(* Version history:
Date	|	Version/Author |	Remark
----------------------------------------------------------------------------------------------------
11.09.01	|	2.01 JP		|	new version depending on 0.99D
22.11.01	|	2.02 JP		|	new version depending on 0.99F
18.01.02	|	2.03 JP		|	new version depending on 1.0
		|				|	changed names, interfaces, execute behavior
25.01.02	|	2.04 JP		|	no CAMMING, change behavior of MC_Power
07.02.02	|	2.05 JP		|	SetOverride in unit less than 1%
13.02.02	|	2.06 JP		|	New: MC_NewPos and MC_NewPosAndVelo
		|				|	removed MC_MoveAdditive
14.02.02	|	2.07 JP		|	completed: MC_Home, MC_MoveSuperImposed
14.02.02	|	2.08 JP		|	renamed MC_NewPosAndVelo New: MC_SetOverride edge triggered
15.02.02	|	2.09 JP		|	changed: MC_Gear
15.02.02	|	2.10 JP		|	changed: MC_SetOverride
04.04.02	|	2.11 JP		|	changed: done for MC_Home 
		|				|	new: Check TimeOut for MoveAbsolute, MoveRelative, Home
08.03.02	|	2.12 JP		|	changed: new flag inserted 
12.03.02	|	2.13 JP		|	changed: reset of bNotExecute
18.03.02	|	2.14 JP		|	changed: MC_Reset waits for ready
22.03.02	|	2.15 JP		|	changed: MC_Read and Write FBs
26.03.02	|	2.16 JP		|	revised: Read/Write Parameter FBs
27.03.02	|	2.17 JP		|	revised: Read/Write Parameter FBs and Home (calibration cam)
09.04.02	|	2.18 JP		|	changed parameter type of some parameters
17.04.02	|	2.19 JP		|	changed: Read(Bool)Parameter new Input to select read mode
							Boolean parameters can be read with ReadParameter
							changed MC_Power: new input override !!			
23.04.02	|	2.20 JP		|	fixed: MC_Home changed: Behavior of MC_MoveAbsolute/Relative
25.04.02	|	2.21 JP		|	changed: MC_Reset: now not waiting for 'axis is ready'. Check with MC_Power !
26.04.02	|	2.22 JP		|	MC_Home: If Posistion =  DEFAULT_HOME_POSITION --> no set of position
							MC_MoveXX: more detailed error messages
05.07.02	|	2.23 JP		|	new MC_MoveAbsoluteOrRestart: combines MoveAbsolute and NewPos
19.07.02	|	2.24 JP		|	changed: E_STATES ---> E_TCMC_STATES
12.09.02	|	2.25 KST		|	changed: MC_MoveAbsolute and MC_MoveRelative now based on FB_MoveGeneric
							MC_NewPos and MC_NewPosAndVelo based on new FB_NewPosAndVeloGeneric 
							new internal start types in MC_MoveAbsoluteOrRestart (message suppression)
16.09.02	|	2.26 ChristophC|	changed: MC_SetActualPosition due to changes in TcNC.Lib
16.10.02	|	2.27 KST		|	new: MC_ExtSetPointGenEnable and MC_ExtSetPointGenDisable
29.10.02	|	2.28 ChristophC|	MC_Stop and MC_SetActualPosition: Ads port changed from TcMcGlobal.NCPORT_TCMC => AMSPORT_R0_NCSAF
12.11.02	|	2.29 ChristophC|	MC_OverrideFilter function block added
13.12.02	|	2.30 JP		|	several smaller changes: MC_ReadStatus, MC_Stop
22.01.03	|	2.31 KSt		|	new additional function MC_ExtSetPointGenFeed
24.03.03	|	2.32 JP		|	added: MC_GearFloat, corr. MC_ReadBoolParameter (wrong for AxisEnPostionRangeMonitoring)
26.03.03	|	2.33 KSt		|	added: MC_MoveModulo
04.04.03	|	2.34 KSt		|	changed: MC_MoveAbsoluteOrRestart, Done will be reset at once after Execute=FALSE
12.05.03	|	2.35 JP		|	changed: MC_MoveVelocity, MC_Home (error handling), MC_ReadStatus
14.05.03	|	2.36 KSt		|	changed: MC_Home, MC_MoveAbsoluteOrRestart
15.05.03	|	2.36.1 KSt	|	changed: MC_Home
28.05.03	|	2.37 KSt		|	changed: MC_MoveVelocity, abort during acceleration phase	
							changed: MC_MoveAbsoluteOrRestart, reset internal error on restart
27.06.03	|	2.38 JP		|	changed: MC_Stop: Execute behavior
22.07.03	|	2.38.1 KSt	|	added: new error codes
12.08.03	|	2.39 KSt		|	changed: FB_ReadWriteParameter, size of bool parameters
15.08.03	|	2.40 KSt		|	added: new block MC_ChangeDynParam
19.08.03	|	2.41 JP		|	changed: MC_ReadParameter: Done falls with Execute
01.10.03	|	2.42 KSt		|	changed: MC_MoveAbsoluteOrRestart, Execute directly after done issue fixed
09.10.03	|	2.43 KSt		|	new function block MC_SetReferenceFlag
04.12.03	|	2.44 KSt		|	ReadBoolParameter(AxisEnTargetPositionMonitoring) corrected
12.01.04	|	2.45 KSt		|	MC_MoveSuperimposed revised
						|	R_Trigger(execute) moved outside CASE in all move function blocks
19.01.04	|	2.45.1 KSt	|	Busy Signal in MC_MoveSuperimposed
30.04.04	|	2.46.0 KSt	|	New function blocks MC_TouchProbe, MC_AbortTrigger, internal block MC_OrientedStop
						|	MC_ReadParameter revised
06.05.04	|	2.46.1 KSt	|	Correction in MC_OrientedStop
21.05.04	|	2.47.0 KSt	|	MC_GearInDyn added - master slave coupling with dynamic gear ratio
06.08.04	|	2.47.1 KSt	|	MC_OrientedStop moved from internal to additional folder
						|	MC_MoveAbsoluteOrRestart additional internal error code NC_ERROR_STARTINTERNAL_NOTREADY evaluated
23.08.04	|	2.47.2 KSt	|	new local flag EmergencyStop in MC_Stop signals type of internal ADS stop command
10.01.05	|	2.47.3 KSt	|	new function block MC_MoveSuperImposedExt
28.01.05	|	2.47.4 KSt	|	TcMcGlobal.tTargetPosTimeOut changed from 5 sec to 6 sec to be later than a NC PEH error (5 sec)
15.02.05	|	2.48.0 KSt	|	new function block MC_GearOutExt 
28.02.05	|	2.49.0 JP		|	Execute and Done behavior corrected for MC_ReadActualPos and MC_SetActualPos
10.03.05	|	2.50.0 KSt	|	all function blocks use a global AMS net-ID TcMcGlobal.NCNETID_TCMC which may be modified by the user
17.03.05	|	2.51.0 KSt	|	new function block MC_PowerStepper
						|	MC_MoveAbsoluteOrRestart restart while starting (adswrite.Busy) changed
24.05.05	|	2.52.0 KSt	|	acceleration added to block MC_GearOutExt 
05.07.05	|	2.53.0 KSt	|	new local flag ADSbusy in all function blocks
05.07.05	|	2.54.0 KSt	|	new function block MC_GearInDynCCV
06.07.05	|	2.55.0 KSt	|	Busy timing improved in all function blocks (turns immediately to FALSE with Done or Error or Aborted)
25.07.05	|	2.55.1 KSt	|	Change for status output behavior 
26.07.05	|	2.55.2 KSt	|	MC_GearOutExt extended through mode 'oriented stop'
03.08.05	|	2.55.3 KSt	|	Commands MC_MoveAbsoluteOrRestart, MC_NewPos and MC_NewPosAndVelo now directed to port AMSPORT_R0_NCSAF
						|	Summary of other commands to SAF: MC_Stop, MC_OrientedStop, MC_TouchProbe, MC_AbortTrigger, MC_SetReferenceFlag, MC_PowerStepper
14.09.05	|	2.56.0 KSt	|	new function block MC_ParameterizedStop
26.09.05	|	2.56.1 KSt	|	Jerk parameter added to MC_ChangeDynParam. Block moved into the internal folder.
07.11.05	|	2.56.2 KSt	|	internal block FB_ReadCharacteristicValues changed to ADSRDWRT
19.12.05	|	2.56.3 KSt	|	new block MC_SetActualPositionOnTheFly
05.01.06	|	2.56.4 KSt	|	new blocks MC_ReadParameterSet and MC_ReadAxisComponents
21.02.06	|	2.57.0 KSt	|	NC status feedback monitoring changed in MC_GearIn and MC_GearInFloat
29.03.06	|	2.57.1 KSt	|	new order of the blocks in the library tree
11.04.06	|	2.57.2 HKP	|	Command MC_ChangeDynParam now directed to port AMSPORT_R0_NCSAF
10.05.06	|	2.57.3 KSt	|	new function block MC_Jog
17.05.06	|	2.57.4 KSt	|	MC_Jog: MC_JOGMODE_INCHING_MODULO temporarily deactivated
05.07.06	|	2.57.5 KSt	|	NC status feedback monitoring changed in MC_GearInDyn and MC_GearInDynCCV
=======	|===============	|==========================================================================
12.07.06	|	2.57.6 KSt	|	new AMS port NCPORT_TCMC_COUPLING for all coupling commands
11.08.06	|	2.57.7 KSt	|	reset Done when Execute is FALSE in FB_NewPosAndVeloGeneric
						|	MC_Jog released
22.08.06	|	2.57.8 KSt	|	new function block MC_AbortSuperposition
07.11.06	|	2.57.9 HKP	|	changes in function block MC_PowerStepper
06.02.07	|	2.57.10 KSt	|	initialization problem with modulo positions fixed in MC_TouchProbe.
						|	recorded position at PlcEvent now modulo when requested.
14.03.07	|	2.57.11 KSt	|	MC_Jog: Handling of CommandAborted corrected
24.04.07	|	2.57.12 KSt	|	additional parameters in MC_AxisPara, MC_ReadParameters, MC_WriteParameters
31.05.07	|	2.57.13 KSt	|	FPU exception with LREAL_TO_BOOL and DWORD_TO_BOOL fixed in FB_ReadWriteParameter 
12.06.07	|	2.57.14 KSt	|	FB_NewPosAndVeloGeneric and MC_MoveSuperImposed(Ext): IF condition changed from "NOT AxisIsMoving" to "NOT AxisHasJob"
=======	|===============	|==========================================================================
12.06.07	|	2.57.14 KSt	|	TcMC2 development started - following 2.xx.xx changes have been added in parallel
02.11.07	|	2.57.15 KSt	|	data structure ST_TableCharacValues extended
18.12.07	|	2.57.16 KSt	|	MC_Jog is now internally using MC_MoveRelative instead of MC_MoveAbsolute to work with backlash compensation
20.05.08	|	2.57.18 KSt	|	AxisModuloPositionFlag added to MC_ReadBoolParameter
17.06.08	|	2.57.20 KSt	|	MC_GearInMultiMaster added
24.07.08	|	2.57.22 KSt	|	MC_Power supports now a minimum Enable-Off/On toggle time of 50ms to reenable the Status output
28.10.08	|	2.57.23 KSt	|	new function block MC_SetEncoderScalingFactor
=======	|===============	|==========================================================================
16.03.07	|	3.00.00 KSt	|	new version depending on PLCopen V1.1 (beta)
25.08.08   |	3.00.01 KSt	|	released as TcMC2 
17.09.08   |	3.00.02 KSt	|	last result added in MC_Reset
26.11.08   |	3.00.03 KSt	|	change in MC_Stop and MoveGeneric for delayed error handling
01.12.08   |	3.00.04 KSt	|	MC_Stop - Done is set immediately at standstill
18.12.08   |	3.00.05 KSt	|	MC_Power - uses now ControlLoopClosed instead of AxisIsReady
13.01.09   |	3.00.06 KSt	|	independent characteristic data for camming and flying saw
16.01.09   |	3.00.07 KSt	|	all move commands: changed handling of CmdNo=0 and CmdNo+2 leads to better results (CommandAborted)
23.01.09   |	3.00.08 KSt	|	MC_MoveSuperimposed is now passed to port AMSPORT_R0_NCSAF (501)
28.01.09   |	3.00.09 KSt	|	Homing mode MC_Direct added - Mode option for MC_SetPosition added
29.01.09   |	3.00.10 KSt	|	Warning output added to MC_MoveSuperimposed
05.02.09   |	3.00.11 KSt	|	axis state is now DISABLED if control loop is not closed (was STANDSTILL for virtual axes - _F_AxisState)
05.02.09   |	3.00.11 KSt	|	all move commands: CmdNo=0 is ignored as invalid - change of the coupled state leads to CommandAborted
06.02.09   |	3.00.11 KSt	|	errors on missing cyclic NC command feedback are delayed for a few cycles to avoid problems with multiple function block calls during one PLC cycle
19.02.09   |	3.00.12 KSt	|	MC_GearInDyn and MC_GearInMultimaster - no reset of gear ratio after Enable is reset to FALSE
24.02.09   |	3.01.00 KSt	|	Motion commands on slaves (must be enabled in the axis parameters before)
12.03.09   |	3.01.01 KSt	|	MC_Jog - Active output added - reset outputs when Execute is false 
09.04.09   |	3.01.02 KSt	|	MC_SetPosition and MC_SetEncoderScalingFactor - explicit encoder / control loop index 0..n can be selected
15.04.09   |	3.01.03 KSt	|	MC_Stop - outputs (except Busy) are reset after Execute=FALSE - can be retriggered during release phase
17.04.09   |	3.01.04 KSt	|	MC_Home - static homing with DEFAULT_HOME_POSITION implemented - Option.ClearPositionLag available 
11.05.09   |	3.01.05 KSt	|	MC_Stop - incorrect error message 4B63 removed;  
30.06.09   |	3.01.06 KSt	|	MC_MoveSuperimposed - new types ACCREDUCTION - new AbortOptions
28.07.09   |	3.01.07 KSt	|	MC_ExtSetPointGenFeed feeds additional counter information to the NC
13.08.09   |	3.01.08 KSt	|	MC_MoveSuperimposed - new AbortOptions - Done behavior adapted
01.09.09   |	3.01.09 KSt	|	MC_SetPosition - new option 'set absolute measuring'
30.09.09   |	3.01.10 KSt	|	MC_MoveSuperimposed - fix for new AbortOptions - HasJob flag not required before starting the command
06.10.09   |	3.01.11 KSt	|	MC_Stop - wait extra cycles before axis release error 
06.10.09   |	3.01.12 KSt	|	MC_MoveSuperimposed - fix for new AbortOptions - HasJob or IsMoving check at beginning and end of compensation 
07.10.09   |	3.01.13 KSt	|	MC_MoveSuperimposed - initial motion check removed for new AbortOptions
28.10.09   |	3.01.14 KSt	|	MC_ExtSetPointGenEnable/Disable - port changed from SVB to SAF
06.11.09   |	3.01.15 KSt	|	MC_SetPosition - new option 'set absolute measuring' removed
09.11.09   |	3.01.16 KSt	|	MC_Stop on slave axes was not rejected with error - fixed
18.11.09   |	3.01.17 KSt	|	MC_Jog - usage with protected (coupled) axes refused
26.11.09   |	3.01.18 KSt	|	Axis status data: UpdateCycleTime calculation fixed
08.12.09   |	3.01.19 KSt	|	_FB_MoveGeneric - mapping check to avoid early Error and CommandAborted signals
25.02.10   |	3.01.20 KSt	|	MC_MoveSuperimposed - additional outputs ActualAcceleration and ActualDeceleration
11.03.10   |	3.01.21 KSt	|	MC_Power - no Enable timeout error for coupled axes
07.04.10   |	3.01.22 KSt	|	MC_ReadApplicationRequest added
15.04.10   |	3.01.23 KSt	|	MC_PositionCorrectionLimiter added - cyclic update of UpdateTaskIndex and UpdateCycleTime removed from ReadStatus
23.04.10   |	3.01.24 KSt	|	internal MC_TouchProbe_V2_00 for new multi probe interface
04.05.10   |	3.01.25 KSt	|	fix in MC_WriteParameter to write bool parameters with MC_WriteParameter as well as MC_WriteBoolParameters
06.05.10   |	3.01.25 KSt	|	fix in MC_MoveContinous... for output InEndVelocity
31.05.10   |	3.02.00 KSt	|	_TcMC_ADS commands added to allow PLC running faster than NC, added to MC_Reset
08.07.10   |	3.02.01 KSt	|	fix in NC mapping counter monitoring (time-out check)
24.09.10   |	3.02.02 KSt	|	ST_NcApplicationRequest structure extended
27.10.10   |	3.02.03 KSt	|	MC_TouchProbe - TRUNC function replaced by MODABS for modulo calculations
22.11.10	|	3.02.04 KSt	|	MC_Power - axis will be enabled automatically after Error turns to FALSE and control loop is closed (just if Enable=TRUE)
		|				|	Move-Commands on axes with external set point generator (must be enabled in the axis parameters before)
29.11.10	|	3.02.05 KSt	|	MC_ReadParameter - new parameters AxisCycleTime NcSafCycleTime and NcSvbCycleTime
17.01.11	|	3.02.06 KSt	|	Phasing blocks added
21.01.11	|	3.02.06 KSt	|	MC_ExtSetPointGenEnable and MC_ExtSetPointGenDisable: code rewritten in ST
16.02.11	|	3.02.07 KSt	|	MC_TouchProbe and MC_TouchProbe_V2_00 - correction for WindowOnly with FirstPosition>LastPosition
18.02.11	|	3.02.08 KSt	|	MC_TouchProbe_V2_00 - TRIGGER_REF extended by optional physical input definition 
21.02.11	|	3.02.08 KSt	|	_MC_Phasing beta version included
25.03.11	|	3.02.09 KSt	|	minor adaption to PlcOpen V2.0 "Function blocks for motion control" released document.
05.04.11	|	3.02.10 KSt	|	new parameters defined for fast axis stopp 
21.04.11	|	3.02.11 KSt	|	FB_MoveUniversalGeneric - fix in command number overrun calculation 
27.04.11	|	3.02.12 KSt	|	new function block MC_ReadStopInfo to read the expected distance and time to stop an axis
02.05.11	|	3.02.13 KSt	|	dynamical data for fast axis stopp can be read or written by MC_ReadParameter, MC_WriteParameter
03.05.11	|	3.02.14 KSt	|	MC_TouchProbe_V2_00 - additional output data structure MC_TouchProbeRecordedData 
11.05.11	|	3.02.15 KSt	|	type check adaptions for the PLC3 compiler
18.05.11	|	3.02.16 KSt	|	data types ST_AxisParameterSet and ST_NcApplicationRequest extended
31.05.11	|	3.02.17 HKP	|	Check of AxisIsReady removed from MC_MoveCommands
31.05.11	|	3.02.17 KSt	|	Axis.OpMode.SimulationAxis added
29.06.11	|	3.02.18 KSt	|	MC_ReadParameterSet fixed for use with differently aligned systems (ARM)
12.07.11	|	3.02.19 KSt	|	internal storage added to AXIS_REF
19.07.11	|	3.02.20 KSt	|	Two Speed Axes: InVelocity detection fixed in MC_MoveVelocity
01.08.11	|	3.02.21 KSt	|	Check of cyclic motion command call - 'buffered command monitoring error' changed to 'cyclic call error' if not cyclically called
07.09.11	|	3.02.22 KSt	|	optional advanced slave motion profile for MC_GearInMultiMaster
13.10.11	|	3.02.23 KSt	|	new OpMode flag AllowExtSetAxisCommands
08.12.11	|	3.02.25 KSt	|	stop monitoring for stop and halt commands added (comparable with target position monitoring)
22.12.11	|	3.02.26 KSt	|	MC_Reset fixed for short PLC cycle times (_TcMC_ADSWRITE waits 2 cycles for NC process image)
22.12.11	|	3.02.27 KSt	|	MC_GearOut and MC_CamOut are now waiting for the NC couple state feedback in Nc2Plc
19.01.12	|	3.02.28 KSt	|	MC_TouchProbe_V2 released
23.02.12	|	3.02.29 ICh	|	_ST_TcNc_OperationModes: cleanup, StopMonitoring added, _ST_TcNC_SetPos: fReserved added to match NC definition
23.02.12	|	3.02.30 KSt	|	typecasts for TC3 to avoid TC3 compiler messages
23.03.12	|	3.02.31 KSt	|	initialization code for MoveModulo revised 
16.05.12	|	3.02.32 KSt	|	MC_MoveVelocity: InVelocity is now reset after abortion or error
05.07.12	|	3.02.33 KSt	|	state diagram changed - if axis has error, state is always ERRORSTOP (never DISABLED)
27.07.12	|	3.02.34 KSt	|	new function blocks MC_BacklashCompensation and MC_TableBasedPositionCompensation. MC_PositionCorrectionLimiter: Acceleration=0 means disables limitation.
23.08.12	|	3.02.35 KSt	|	MC_Power now avoids time out errors after an axis reset
04.04.13	|	3.02.36 KSt	|	extended ST_DriveAddress structure; used with MC_ReadDriveAddress
02.07.13	|	3.02.37 KSt	|	Done may have come together with Error or CommandAborted - fixed by resetting Done in these cases.
10.07.13	|	3.02.38 KSt	|	MC_Move commands now check NC interface update before monitoring NC feedback
02.09.13	|	3.02.39 KSt	|	MC_PositionCorrectionLimiter - mode UNLIMITED for axes in standstill fixed (was internally set to FAST before)
04.09.13	|	3.02.40 KSt	|	now waiting for READDEVINFO (NC version) in MC_AbortTrigger_V2_00 and MC_ReadDriveAddress
01.10.13	|	3.02.41 KSt	|	function MC_SetAcceptBlockedDriveSignal added
01.10.13	|	3.02.42 KSt	|	debug message for positive move commands can be enabled with ControlDWord.29
22.11.13	|	3.02.43 KSt	|	Avoid too early Active output at Move commands - now waiting for NcToPlc mapping after ADS command
21.03.14	|	3.02.44 KSt	|	MC_AbortTrigger now falls back to initialization state and resets busy after operration
20.05.14	|	3.02.45 KSt	|	correction of Status.UpdateCycleTime in _F_ReadStatus
14.07.14	|	3.02.46 KSt	|	MC_ReadParameter, MC_WriteParameter, Port changed to 501 for parameters AxisRemainingTimeToGo and AxisRemainingDistanceToGo
22.10.14	|	3.02.47 KSt	|	MC_Move commands Active feedback optimized. Active now turns to true as soon as the CmdNo has definitely changed and is equal to own number (NC response).
23.10.14	|	3.02.48 KSt	|	MC_BacklashCompensation - Correction in parameter check
30.09.14	|	3.02.49 KSt	|	MC_MoveSuperimposed and MC_AbortSuperposition now redirected to NCPORT_TCMC_SUPERPOSITION, port can be modified by user
19.03.15	|	3.02.50 KSt	|	MC_Stop command can now be aborted by a reset command if axis is in standstill and the flag "Motion Commands Locked" is false
05.05.15	|	3.02.51 KSt	|	MC_Power - error feedback in case of axis errors corrected 
19.10.15	|	3.02.52 FAp	|	optimization for MC_GearInMultiMaster

*)
CASE nVersionElement OF
1:	(* major number *)
	F_GetVersion_TcMC2 := 3;
2:	(* minor number *)
	F_GetVersion_TcMC2 := 2;
3:	(* revision number *)
	F_GetVersion_TcMC2 := 52;
ELSE
	F_GetVersion_TcMC2 := 16#FFFF;
END_CASE
END_FUNCTION

(* POU MC_AbortSuperposition, ST *)
FUNCTION_BLOCK MC_AbortSuperposition
VAR_INPUT
	Execute		:	BOOL;	(* Starts touch probe recording *)
END_VAR
VAR_OUTPUT
	Done		:	BOOL;	(* move completed *)
	Busy		: 	BOOL;	(* function block is currently Busy *)
	Error		:	BOOL;	(* Signals that error has occured within Function Block *)
	ErrorID		:	UDINT;	(* Error identification *)
END_VAR
VAR_IN_OUT
	Axis			:	AXIS_REF; (* Identifies the axis of which the position should be recorded at a defined event at the trigger input *)
END_VAR
VAR
	LastExecutionResult: 	_ST_FunctionBlockResults;
	ADSbusy	: 	BOOL;
	fbOnTrigger	: 	R_TRIG;
	fbADSwrite	: 	ADSWRITE;
	iState		:	_E_TcMC_STATES := STATE_INITIALIZATION;
END_VAR
fbOnTrigger(CLK:= Execute);

CASE iState OF
STATE_INITIALIZATION: (* initial iState *)
	Busy := FALSE;
	IF NOT Execute THEN
		Done := FALSE;
		Error := FALSE;
		ErrorID := 0;
	END_IF
	IF fbOnTrigger.Q THEN
		Busy := TRUE;
		(* initialization *)
		Done := FALSE;
		Error := FALSE;
		ErrorID := 0;
		LastExecutionResult.Done := FALSE;
		LastExecutionResult.CommandAborted := FALSE;
		LastExecutionResult.Error := FALSE;
		LastExecutionResult.ErrorID := 0;
		fbADSwrite(WRITE:=FALSE);
		fbADSwrite(	NETID:= TcMcGlobal.NCNETID_TCMC,
					(* PORT:=TcMcGlobal.NCPORT_TCMC , *)		(* 20140930 KSt *)
					PORT:=TcMcGlobal.NCPORT_TCMC_SUPERPOSITION,	(* 20140930 KSt *)
					IDXGRP:= TcMcGlobal.Axis.Functions.IDXGRP + Axis.NcToPlc.AxisId,
					IDXOFFS:= TcMcGlobal.Axis.Functions.IDXOFFS.STOPSCOM,	(* abort superposition *)
					LEN:=0,
					SRCADDR:=0,
					WRITE:=TRUE ,
					TMOUT:= TcMcGlobal.tADSTimeOut);
		iState := STATE_ORDER;
	END_IF

STATE_ORDER:  (* wait until command is accepted *)
	fbADSwrite(WRITE:= TRUE);
	IF NOT fbADSwrite.BUSY THEN
		Error := fbADSwrite.ERR;
		ErrorID := fbADSwrite.ERRID;
		IF NOT Error THEN
			IF NOT F_AxisIsCompensating(Axis.NcToPlc.StateDWord) THEN
				Done := TRUE;
				Busy := FALSE;
				iState := STATE_INITIALIZATION;
			ELSE
				iState := STATE_RUNNING;
			END_IF
		ELSE
			Busy := FALSE;
			iState := STATE_INITIALIZATION;
		END_IF
		LastExecutionResult.Done := Done;
		LastExecutionResult.Error := Error;
		LastExecutionResult.ErrorID := ErrorID;
	END_IF

STATE_RUNNING:
	IF NOT F_AxisIsCompensating(Axis.NcToPlc.StateDWord) THEN
		Done := TRUE;
		Busy := FALSE;
		LastExecutionResult.Done := Done;
		LastExecutionResult.Error := Error;
		LastExecutionResult.ErrorID := ErrorID;
		iState := STATE_INITIALIZATION;
	END_IF
END_CASE

ADSbusy := fbAdsWrite.BUSY;
END_FUNCTION_BLOCK

(* POU MC_AbortTrigger, ST *)
FUNCTION_BLOCK MC_AbortTrigger
(*	The function block is used to abort function blocks which are connected to
	trigger events (e.g. MC_TouchProbe) 
*)
VAR_IN_OUT
	Axis			:	AXIS_REF; 		(* B *)	(* Identifies the axis of which the position should be recorded at a defined event at the trigger input *)
	TriggerInput	: 	TRIGGER_REF; 	(* E *)	(* Reference to the trigger signal source. *)
END_VAR
VAR_INPUT
	Execute		:	BOOL;	(* B *)	(* Starts aborting  touch probe sequence *)
END_VAR
VAR_OUTPUT
	Done		:	BOOL;	(* B *)	(* function completed *)
	Busy		: 	BOOL;	(* E *)	(* function block is currently Busy *)
	Error		:	BOOL;	(* B *)	(* Signals that error has occurred within Function Block *)
	ErrorID		:	UDINT;	(* E *)	(* Error identification *)
END_VAR
VAR
	ADSbusy	: 	BOOL;
	fbADSwrite	: 	ADSWRITE;
END_VAR
{library private}
VAR CONSTANT
	OLDADSINTERFACE : BOOL := TRUE; (* temporary flag to test old and new NC ADS touch probe interface *)
END_VAR
VAR
	LatchID		: 	UDINT;
	fbOnTrigger	: 	R_TRIG;
END_VAR
IF NOT Execute THEN
	Done := FALSE;
	Error := FALSE;			(* reset at falling edge of Execute *)
	ErrorID := 0;
END_IF

fbOnTrigger(CLK:= Execute);
IF fbOnTrigger.Q OR fbADSwrite.BUSY THEN
	Busy := TRUE;
	IF fbOnTrigger.Q THEN
		(* initialization *)
		Done := FALSE;
		Error := FALSE;
		ErrorID := 0;
		fbADSwrite(WRITE:=FALSE);
		IF TriggerInput.EncoderID > 255 THEN
			Error := TRUE;
			ErrorID := MC_ERROR_INVALID_TOUCH_PROBE;
		END_IF
	END_IF

	IF NOT Error THEN
		CASE TriggerInput.TouchProbe OF
			TouchProbe1,
			TouchProbe2,
			TouchProbe3,
			TouchProbe4:
			LatchID := TriggerInput.TouchProbe;
			fbADSwrite(	NETID:= TcMcGlobal.NCNETID_TCMC,
						PORT:=AMSPORT_R0_NCSAF ,
						IDXGRP:=16#5200+TriggerInput.EncoderID ,
						IDXOFFS:=16#205,	(* deactivate touch probe *)
						LEN:=SEL(OLDADSINTERFACE, SIZEOF(LatchID), 0) ,
						SRCADDR:=ADR(LatchID),
						WRITE:=TRUE ,
						TMOUT:=TcMcGlobal.tADSTimeOut);
			IF NOT fbADSwrite.BUSY THEN
				Error := fbADSwrite.ERR;
				ErrorID := fbADSwrite.ERRID;
				TriggerInput.ProbeState := SEL(Error, TouchProbeAborted, TriggerInput.ProbeState );
				Done := NOT Error;
			END_IF

			PlcEvent:
				(* no action necessary here *);
				TriggerInput.ProbeState := TouchProbeAborted;
				Done := TRUE;

			ELSE (* case *)
				Error := TRUE;
				ErrorID := MC_ERROR_INVALID_TOUCH_PROBE;
		END_CASE
	END_IF
ELSE
	Busy := FALSE;
END_IF

ADSbusy := fbAdsWrite.BUSY;
(* reset Busy immediately  when sequence ends *)
Busy := fbOnTrigger.Q OR fbADSwrite.BUSY;
END_FUNCTION_BLOCK

(* POU MC_AbortTrigger_V2_00, ST *)
FUNCTION_BLOCK MC_AbortTrigger_V2_00
(*	The function block is used to abort function blocks which are connected to
	trigger events (e.g. MC_TouchProbe) 
*)
VAR_IN_OUT
	Axis			:	AXIS_REF; 		(* B *)	(* Identifies the axis of which the position should be recorded at a defined event at the trigger input *)
	TriggerInput	: 	TRIGGER_REF; 	(* E *)	(* Reference to the trigger signal source. *)
END_VAR
VAR_INPUT
	Execute		:	BOOL;	(* B *)	(* Starts aborting  touch probe sequence *)
END_VAR
VAR_OUTPUT
	Done		:	BOOL;	(* B *)	(* function completed *)
	Busy		: 	BOOL;	(* E *)	(* function block is currently Busy *)
	Error		:	BOOL;	(* B *)	(* Signals that error has occurred within Function Block *)
	ErrorID		:	UDINT;	(* E *)	(* Error identification *)
END_VAR
VAR
	ADSbusy	: 	BOOL;
	fbADSwrite	: 	ADSWRITE;
	i: INT;
	iState			: 	_E_TcMC_STATES := STATE_INITIALIZATION;
END_VAR
{library private}
VAR
	LatchID		: 	UDINT;
	fbOnTrigger	: 	R_TRIG;
	stTouchProbeDeactivation : _ST_TcNc_TouchProbeDeactivation;
END_VAR
IF NOT Execute THEN
	Done := FALSE;
	Error := FALSE;			(* reset at falling edge of Execute *)
	ErrorID := 0;
END_IF

fbOnTrigger(CLK:= Execute);

FOR i := 1 TO 2 DO (* typically aborted after one scan *)
	CASE iState OF
		STATE_INITIALIZATION :

			IF fbOnTrigger.Q OR fbADSwrite.BUSY THEN
				Busy := TRUE;

				IF fbOnTrigger.Q THEN
					(* initialization *)
					Done := FALSE;
					Error := FALSE;
					ErrorID := 0;
					fbADSwrite(WRITE:=FALSE);
					IF TriggerInput.EncoderID > 255 THEN
						Error := TRUE;
						ErrorID := MC_ERROR_INVALID_TOUCH_PROBE;
					END_IF
				END_IF

				IF TcMcGlobal.NcDeviceInfoNcVersion=0 THEN
					(* read version of NC *)
					TcMcGlobal.ReadDeviceInfo();
					iState := STATE_WAITING;
					EXIT; (* FOR loop *)
				ELSIF NOT Error THEN
					iState := STATE_ORDER;
				END_IF
			END_IF

		STATE_WAITING :	(* 2013-09-04 - new waiting state in case of invalid NC version information *)
			(* check for NC version *)
			TcMcGlobal.ReadDeviceInfo();
			IF NOT TcMcGlobal.fbADSRDDEVINFO.BUSY THEN
				istate := STATE_ORDER;
			ELSE
				EXIT; (* FOR loop *)
			END_IF

		STATE_ORDER :
			CASE TriggerInput.TouchProbe OF
				TouchProbe1,
				TouchProbe2,
				TouchProbe3,
				TouchProbe4:
					IF TcMcGlobal.NcDeviceInfoNcVersion > 16#020B07DD AND (TriggerInput.mode<>TOUCHPROBEMODE_SINGLE_COMPATIBILITYMODE) THEN
						(* new touch probe interface since TwinCAT 2.11 Nc-Driver 2014 *)
						stTouchProbeDeactivation.TouchProbe := TriggerInput.TouchProbe;
						stTouchProbeDeactivation.Edge := TriggerInput.Edge;
						fbADSwrite(	NETID:= TcMcGlobal.NCNETID_TCMC,
									PORT:=AMSPORT_R0_NCSAF ,
									IDXGRP:=16#5200+TriggerInput.EncoderID ,
									IDXOFFS:=16#205,	(* deactivate touch probe *)
									LEN:= SIZEOF(stTouchProbeDeactivation),
									SRCADDR:=ADR(stTouchProbeDeactivation),
									WRITE:=TRUE ,
									TMOUT:=TcMcGlobal.tADSTimeOut);
					ELSE
						(* classic touch probe interface *)
						fbADSwrite(	NETID:= TcMcGlobal.NCNETID_TCMC,
									PORT:=AMSPORT_R0_NCSAF ,
									IDXGRP:=16#5200+TriggerInput.EncoderID ,
									IDXOFFS:=16#205,	(* deactivate touch probe *)
									LEN:= 0,
									SRCADDR:=0,
									WRITE:=TRUE ,
									TMOUT:=TcMcGlobal.tADSTimeOut);
					END_IF
					IF NOT fbADSwrite.BUSY THEN
						Error := fbADSwrite.ERR;
						ErrorID := fbADSwrite.ERRID;
						TriggerInput.ProbeState := SEL(Error, TouchProbeAborted, TriggerInput.ProbeState );
						Done := NOT Error;
						iState := STATE_INITIALIZATION;	(* 2014-03-21 KSt *)
					END_IF

				PlcEvent:
					(* no action necessary here *);
					TriggerInput.ProbeState := TouchProbeAborted;
					Done := TRUE;
					iState := STATE_INITIALIZATION;	(* 2014-03-21 KSt *)

				ELSE (* case *)
					Error := TRUE;
					ErrorID := MC_ERROR_INVALID_TOUCH_PROBE;
					iState := STATE_INITIALIZATION;	(* 2014-03-21 KSt *)
			END_CASE
			EXIT; (* FOR loop *)
END_CASE
END_FOR

ADSbusy := fbAdsWrite.BUSY;
IF iState=STATE_INITIALIZATION THEN
	(* reset Busy immediately  when sequence ends *)
	Busy := FALSE;
END_IF
END_FUNCTION_BLOCK

(* POU MC_BacklashCompensation, ST *)
(*==============================================================================*)
(* Name:	MC_BacklashCompensation												*)
(*		(based on _FB_PositionCorrectionTableLookup + MC_PositionCorrectionLimiter)	*)
(* Parameter: returns a compensation value depending on the position of the reference axis	*)
(*		Use the nc function PositionCompensation to compensate the backlash			*)
(*		1. the FB _FB_PositionCorrectionTableLookup calculates the backlash value		*)
(*		2. the FB MC_PositionCorrectionLimiter feed this correction value					*)
(*		into the NcToPlc.PositionCorrection variable									*)
(* Requirements: The 'Position Correction' feature must be enabled in the SystemManager 	*)
(*																				*)
(* Author:	 	HKP																	*)
(* Date:		19-July-2012															*)
(* last edit:	VER 0.0.4															*)
(*==============================================================================*)

FUNCTION_BLOCK MC_BacklashCompensation
VAR_IN_OUT
	Axis							: Axis_Ref;
END_VAR
VAR_INPUT
	Enable						: BOOL;							(* switch to activate backlash compensation *)
	Backlash					: LREAL := DEFAULT_BACKLASHVALUE;	(* signed backlash value [mm] (when using default value the internal nc backlash value will be read by ADS and used in this FB) *)
	CompensationInPositiveDirection : BOOL;							(* compensation is just working in the selected working direction *)
																(* FALSE (default): backlash compensation must be done when driving in negative direction;  TRUE: backlash compensation must be done when driving in positive direction *)
	Ramp						: LREAL;							(* velocity limit for feeded backlash compensation (constant velocity and linear position sub profile for backlash compensation) [mm/s] (default:=0.0) *)
	DisableMode					: E_DisableMode;					(* disable mode defines whow to react in case of disabling: (0)=HOLD, (1)=RESET, ... *)
	Options						: ST_BacklashCompensationOptions;	(* optional parameters (NOT USED YET) *)
END_VAR
VAR_OUTPUT
	Enabled						: BOOL;
	Busy						: BOOL;
	Error						: BOOL;
	ErrorID						: UDINT;
	CurrentBacklash				: LREAL;							(* current actual backlash value [mm] *)
	Limiting						: BOOL;							(* function block is currently limiting the Backlash Correction *)
END_VAR
VAR
	InternalEnable				: BOOL;							(* trick for internal FB handling *)
	state						: INT;
	GetThisTaskIndex				: GETCURTASKINDEX;
	CycleTime					: LREAL;								(* task cycle time [s] *)
	fbCalcBacklashCorrection		: _FB_PositionCorrectionTableLookup;	(* based on old 'FB_PositionCompensation' in TcNc.lib *)
	fbFeedBacklashCorrection		: MC_PositionCorrectionLimiter;			(* s.TcMC2.lib (original based on old 'FB_WritePositionCorrection' in TcNc.lib) *)
	CalcBacklashCorrOut			: ST_McOutputs;
	FeedBacklashCorrOut			: ST_McOutputs;
	ReadParameter				: MC_ReadParameter;
	iBacklash					: LREAL;
	InternalAcceleration			: LREAL;								(* input of FB 'MC_PositionCorrectionLimiter': 'Acceleration' [mm/s^2] *)
	InternalBacklashValue			: LREAL;								(* output of FB 'MC_PositionCorrectionLimiter': 'PositionCorrectionValue' [mm] *)
	InternalLimitingActive			: BOOL;								(* output of FB 'MC_PositionCorrectionLimiter': 'Limiting' [0/1] *)

	stPosCompParameter : ST_PositionCompensationTableParameter :=
								( MinPosition := -1.0E+12, MaxPosition :=1.0E+12, NoOfTableElements :=2, Direction := WorkDirectionNegative );

	stPosCompTable: ARRAY[0..1] OF ST_PositionCompensationTableElement :=
								( Position := -1.0E+12,	Compensation := 0.0 ),
								( Position := +1.0E+12,	Compensation := 0.0 );
END_VAR
CASE state OF
	0 : (* init *)
		Busy := FALSE;
		Enabled := FALSE;
		IF Enable THEN
			IF NOT Axis.NcToPlc.OpModeDWord.20 THEN (* PositionCorrection active ? *)
				Error := TRUE;
				ErrorID := MC_ERROR_WRONG_MODE;
				state := 9999;
			ELSIF Ramp < 0 THEN
				Error := TRUE;
				ErrorID := MC_ERROR_PARAMETER_NOT_CORRECT;
				state := 9999;
(*			ELSIF Backlash < -100 OR Backlash > 100 THEN *)				(* HKP 2014-10-23 *)
(*				Error := TRUE; *)										(* HKP 2014-10-23 *)
(*				ErrorID := MC_ERROR_PARAMETER_NOT_CORRECT; *)	(* HKP 2014-10-23 *)
(*				state := 9999; *)										(* HKP 2014-10-23 *)
(*			ELSIF Backlash = DEFAULT_BACKLASHVALUE THEN *)		(* HKP 2014-10-23 *)
				(* read default backlash value *)							(* HKP 2014-10-23 *)
(*				ReadParameter( Enable:= FALSE, Axis:= Axis);*)			(* HKP 2014-10-23 *)
(*				Busy := TRUE;*)										(* HKP 2014-10-23 *)
(*				state := 1;*)											(* HKP 2014-10-23 *)
                            ELSIF Backlash = DEFAULT_BACKLASHVALUE THEN	(* HKP 2014-10-23 -  1) ersten auf diesen riesigen Defaultwert prüfen (1.0E307) *)
                                            (* read default backlash value *)
                                            ReadParameter( Enable:= FALSE, Axis:= Axis);
                                            Busy := TRUE;
                                            state := 1;
                            ELSIF Backlash < -100 OR Backlash > 100 THEN		(* HKP 2014-10-23 -  2) erst dann auf sinnvolle User-Eingabe prüfen*)
                                            Error := TRUE;
                                            ErrorID := MC_ERROR_PARAMETER_NOT_CORRECT;
                                            state := 9999;
			ELSE
				iBacklash := Backlash;
				Busy := TRUE;
				state := 10;
			END_IF
		END_IF

	1: (* read default backlash value *)
		ReadParameter(
			Enable:= TRUE,
			ParameterNumber:= AxisBacklash,
			ReadMode:= READMODE_ONCE,
			Axis:= Axis );
		IF ReadParameter.Valid THEN
			iBacklash := ReadParameter.Value;
			IF iBacklash < -100 OR iBacklash > 100 THEN
				Error := TRUE;
				ErrorID := MC_ERROR_PARAMETER_NOT_CORRECT;
				state := 9999;
			ELSE
				state := 10;
			END_IF
		ELSIF ReadParameter.Error THEN
			Error := TRUE;
			ErrorID := ReadParameter.ErrorID;
			state := 9999;
		END_IF

	10 : (* active *)
		Enabled := TRUE;
		(*
		  1.)  Set backlash parameter in dependency of following input parameter: 'CompensationInPositiveDirection' (FALSE/TRUE)
			Remark: The sign of the 'Backlash' value (+/-) doesn't care.
		*)

		(* FALSE (default): backlash compensation must be done when driving in negative direction *)
		IF( NOT CompensationInPositiveDirection ) THEN
			stPosCompParameter.Direction		:= WorkDirectionNegative;
			stPosCompTable[0].Compensation	:= iBacklash;
			stPosCompTable[1].Compensation	:= iBacklash;
		(* TRUE: backlash compensation must be done when driving in positive direction *)
		ELSE
			stPosCompParameter.Direction		:= WorkDirectionPositive;
			stPosCompTable[0].Compensation	:= -iBacklash;
			stPosCompTable[1].Compensation	:= -iBacklash;
		END_IF

		(* BacklashValue = 0.0 *)
		IF ( iBacklash = 0.0 ) THEN
			stPosCompParameter.Direction		:= WorkDirectionNone;
			stPosCompTable[0].Compensation	:= 0.0;
			stPosCompTable[1].Compensation	:= 0.0;
		END_IF


		(* cycle time needed for pre calculation of the acceleration input *)
		IF CycleTime = 0 THEN
			GetThisTaskIndex;
			CycleTime := SystemTaskInfoArr[GetThisTaskIndex.index].cycleTime * LREAL#100E-9;
		END_IF

		(* special handling for disabling (depends from disable mode) *)
		IF( Enable = FALSE ) THEN
			(* disable mode HOLD *)
			IF( (DisableMode = DisableModeHold) ) THEN
				InternalEnable := TRUE;
				IF( Ramp > 0.0 ) THEN
					InternalAcceleration := Ramp / CycleTime;			(* mm/s^2 = mm/s / s *)
				ELSE
					InternalAcceleration := 0.0;
				END_IF
			(* disable mode RESET *)
			ELSE
				InternalEnable := Enable;
				InternalAcceleration := 0.0;
			END_IF
		(* active *)
		ELSE
			InternalEnable := Enable;
			IF( Ramp > 0.0 ) THEN
				InternalAcceleration := Ramp / CycleTime;				(* mm/s^2 = mm/s / s *)
			ELSE
				InternalAcceleration := 0.0;
			END_IF
		END_IF


		(* 2.) calculate backlash correction (if enabled) *)
		(* '_FB_PositionCorrectionTableLookup' *)
		fbCalcBacklashCorrection(
		   (* Enable := Enable, *)
		   Enable := InternalEnable,
		   pTable := ADR(stPosCompTable),
		   TableSize := SIZEOF(stPosCompTable),
		   Axis := Axis,
		   TableParameter := stPosCompParameter,
		   Compensation => InternalBacklashValue,
		   Error => CalcBacklashCorrOut.Error,
		   ErrorId => CalcBacklashCorrOut.ErrorID,
		   Active => CalcBacklashCorrOut.Active );

		(* check for error return code *)
		IF CalcBacklashCorrOut.Error THEN
			Error := TRUE;
			ErrorID := CalcBacklashCorrOut.ErrorID;
			state := 9999;
		END_IF


		(* 3.) feed backlash compensation (acceleration limited, that means linear velocity ramp) *)
		(*
				POSITIONCORRECTIONMODE_FAST
					The limitatation to maximum position change per cycle. Due to the maximum 
					change per cycle, the correction will take place as fast as possible and may 
					also be unlimited if PositionCorrectionValue is changed slightly. 
		*)
		(* MC_PositionCorrectionLimiter *)
		fbFeedBacklashCorrection(
		(*	Enable :=TRUE, *)
			 Enable :=Enable,
			 PositionCorrectionValue := InternalBacklashValue,
			 CorrectionMode := POSITIONCORRECTION_MODE_FAST,
		(*	 Acceleration := BacklashAccelecationLimit, *)	(* HKP: direct feeded user acceleration limit *)
			 Acceleration := InternalAcceleration,			(* HKP: pre calculated internal acceleration limit *)
			 CorrectionLength := 0.0,					(* optional length - not used for this correction mode 'POSITIONCORRECTION_MODE_FAST' *)
			 Axis := Axis,
			 Busy => FeedBacklashCorrOut.Busy,
			 Error => FeedBacklashCorrOut.Error,
			 ErrorID =>FeedBacklashCorrOut.ErrorID,
			 Limiting => InternalLimitingActive
			);

		(* check for error return code *)
		IF FeedBacklashCorrOut.Error THEN
			Error := TRUE;
			ErrorID := FeedBacklashCorrOut.ErrorID;
			state := 9999;
		END_IF


		CurrentBacklash	:= InternalBacklashValue;
		Limiting			:= InternalLimitingActive;

		IF NOT Enable THEN
			Enabled := FALSE;
			state := 0;
		END_IF

	9999 : (* error *)
		IF NOT Enable THEN
			Error := FALSE;
			ErrorID := 0;
			state := 0;
		END_IF
END_CASE

IF state = 0 THEN
	Busy := FALSE;
END_IF
END_FUNCTION_BLOCK

(* POU MC_PositionCorrectionLimiter, ST *)
FUNCTION_BLOCK MC_PositionCorrectionLimiter
(*
 	The function block PositionCorrectionLimiter feed a correction value into the
	NcToPlc.PositionCorrection variable. 

	The correction value corrects the actual position of the encoder. The correction 
	does not only affect the actual position but will also lead to an axis motion caused 
	by the position controller of the axis or drive. The correction does not affect the
	set position of the set-point generator.

	The block supports following modes:
		POSITIONCORRECTIONMODE_UNLIMITED
			no limitation - the PositionCorrectionValue is passed to the NC immediately
		POSITIONCORRECTIONMODE_FAST
			The limitatation to maximum position change per cycle. Due to the maximum 
			change per cycle, the correction will take place as fast as possible and may 
			also be unlimited if PositionCorrectionValue is changed slightly. 
		POSITIONCORRECTIONMODE_FULLLENGTH 
			The limitation uses a defined full CorrectionLength (travel path)  to adapt to 
			the PositionCorrectionValue in small steps. This mode will allways cause a 
			limitation and takes care of a smooth correction.
*)
VAR_IN_OUT
	Axis					:	AXIS_REF;
END_VAR
VAR_INPUT
	Enable				:	BOOL;
	PositionCorrectionValue : 	LREAL;
	CorrectionMode		:	E_AxisPositionCorrectionMode;
	Acceleration			: 	LREAL;
	CorrectionLength		:	LREAL; (* optional length - comparable to 'superposition length' *)
END_VAR
VAR_OUTPUT
	Busy				:	BOOL;
	Error				:	BOOL;
	ErrorID				:	UDINT;
	Limiting				: 	BOOL;	(* function block is currently limiting the Position Correction *)
END_VAR
VAR
	GetThisTaskIndex: GETCURTASKINDEX;
	CycleTime: LREAL;
	MaxDeltaVelocity: LREAL;
	MaxDeltaPosition: LREAL;
	DeltaCorrection: LREAL;
	InitialDeltaCorrection: LREAL;
	EndOfEnablePhase: BOOL;
	iCorrectionMode : E_AxisPositionCorrectionMode;
	state: INT;
	NumberOfCycles: UDINT;
	DeltaCorrectionPerCycle: LREAL;
	LastPositionCorrectionValue: LREAL;
END_VAR
CASE state OF
	0 : (* disabled *)
		Busy := FALSE;
		Limiting := FALSE;
		LastPositionCorrectionValue := 0;
		IF Enable THEN
			(* IF Acceleration<=0 AND CorrectionMode <> POSITIONCORRECTION_MODE_UNLIMITED THEN *) (* KST 20120730 *)
			IF Acceleration<0 AND CorrectionMode <> POSITIONCORRECTION_MODE_UNLIMITED THEN (* KST 20120730 - zero acc means unlimited correction *)
				Error := TRUE;
				ErrorID := MC_ERROR_PARAMETER_NOT_CORRECT;
			ELSIF CorrectionLength <= 0 AND CorrectionMode=POSITIONCORRECTION_MODE_FULLLENGTH THEN
				Error := TRUE;
				ErrorID := MC_ERROR_PARAMETER_NOT_CORRECT;
			ELSE
				Limiting := FALSE;
				Error := FALSE;
				ErrorID := 0;
				state := 1;
				Busy := TRUE;
			END_IF
		ELSE
			Limiting := FALSE;
			Error := FALSE;
			ErrorID := 0;
		END_IF

	1 : (* enabled *)
		Busy := TRUE;
		IF NOT Enable THEN
			state := 2;
		END_IF

	2 : (* disabling *)
		IF Enable THEN
			state := 1;
		ELSE
			PositionCorrectionValue := 0;
			IF Axis.PlcToNc.PositionCorrection = 0 THEN
				state := 0;
			END_IF
		END_IF
END_CASE

CASE state OF
	1, 2:
		IF CycleTime = 0 THEN
			GetThisTaskIndex;
			CycleTime := SystemTaskInfoArr[GetThisTaskIndex.index].cycleTime * LREAL#100E-9;
		END_IF
		MaxDeltaVelocity := Acceleration * CycleTime;
		MaxDeltaPosition := MaxDeltaVelocity * CycleTime;
		DeltaCorrection := PositionCorrectionValue - Axis.PlcToNc.PositionCorrection;

		(* check if correction mode is possible *)
		iCorrectionMode := CorrectionMode;
(*		IF iCorrectionMode=POSITIONCORRECTION_MODE_FULLLENGTH AND CorrectionLength <= 0 OR ABS(Axis.NcToPlc.SetVelo) < 1E-6 THEN *)	(* KSt 2013-09-02 brackets wrong *)
		IF iCorrectionMode=POSITIONCORRECTION_MODE_FULLLENGTH AND (CorrectionLength <= 0 OR ABS(Axis.NcToPlc.SetVelo) < 1E-6) THEN	(* KSt 2013-09-02 brackets new *)
			iCorrectionMode := POSITIONCORRECTION_MODE_FAST;
		END_IF

		CASE iCorrectionMode OF
			POSITIONCORRECTION_MODE_UNLIMITED :
					Limiting := FALSE;
					Axis.PlcToNc.PositionCorrection := PositionCorrectionValue;

			POSITIONCORRECTION_MODE_FAST :
				(* IF ABS(DeltaCorrection) <= MaxDeltaPosition then *) (* KST 20120730 *)
				IF 	ABS(DeltaCorrection) <= MaxDeltaPosition
					OR Acceleration=0 OR MaxDeltaPosition=0 (* KST 20120730 - zero acc means unlimited correction *)
					THEN
					Limiting := FALSE;
					Axis.PlcToNc.PositionCorrection := PositionCorrectionValue;
				ELSE
					Limiting := TRUE;
					IF DeltaCorrection > 0 THEN
						Axis.PlcToNc.PositionCorrection := Axis.PlcToNc.PositionCorrection + MaxDeltaPosition;
					ELSE
						Axis.PlcToNc.PositionCorrection := Axis.PlcToNc.PositionCorrection - MaxDeltaPosition;
					END_IF
				END_IF

			POSITIONCORRECTION_MODE_FULLLENGTH :
				(* check if PositionCorrectionValue changed *)
				(* then calculate the change per cycle and scatter the change over the defined CorrectionLength *)
				IF PositionCorrectionValue<>LastPositionCorrectionValue THEN
					InitialDeltaCorrection := DeltaCorrection;
				END_IF
				LastPositionCorrectionValue := PositionCorrectionValue;
				NumberOfCycles := LREAL_TO_UDINT(CorrectionLength / ABS(Axis.NcToPlc.SetVelo) / CycleTime);
				DeltaCorrectionPerCycle := ABS(InitialDeltaCorrection) / NumberOfCycles;
(*				IF ABS(DeltaCorrectionPerCycle) > MaxDeltaPosition THEN*) (* KST 20120730 *)
				IF 	ABS(DeltaCorrectionPerCycle) > MaxDeltaPosition
					AND MaxDeltaPosition > 0 THEN (* KST 20120730 *)
					DeltaCorrectionPerCycle := MaxDeltaPosition;
				END_IF

				IF ABS(DeltaCorrection) <= DeltaCorrectionPerCycle THEN
					Limiting := FALSE;
					Axis.PlcToNc.PositionCorrection := PositionCorrectionValue;
				ELSE
					Limiting := TRUE;
					IF DeltaCorrection > 0 THEN
						Axis.PlcToNc.PositionCorrection := Axis.PlcToNc.PositionCorrection + DeltaCorrectionPerCycle;
					ELSE
						Axis.PlcToNc.PositionCorrection := Axis.PlcToNc.PositionCorrection - DeltaCorrectionPerCycle;
					END_IF
				END_IF
		END_CASE
END_CASE
END_FUNCTION_BLOCK

(* POU MC_ReadParameter, ST *)
FUNCTION_BLOCK MC_ReadParameter
(*	This Function Block returns the value of a vendor specific parameter *)
VAR_IN_OUT
	Axis				:	AXIS_REF;	(* B *)
END_VAR
VAR_INPUT
	Enable			:	BOOL;		(* B *)
	ParameterNumber	:	INT;			(* B *)
	ReadMode		:	E_ReadMode(* V *) := ReadMode_Once;	 (* Beckhoff proprietary input *)
END_VAR
VAR_OUTPUT
	Valid			:	BOOL;		(* B *)
	Busy			: 	BOOL;		(* E *)
	Error			:	BOOL;		(* B *)
	ErrorID			:	UDINT;		(* E *)
	Value			:	LREAL;		(* B *)
END_VAR
VAR
	ADSbusy		: 	BOOL;
	fbReadWriteParameter: 	_FB_ReadWriteParameter;
END_VAR
{library private}
VAR
	nParatype 		: 	_E_ParameterType;
	dwValue 			: 	DWORD;
	bValue 			: 	BOOL;
	bStarted			:	BOOL;
	fbTrigger		 	: 	R_TRIG;
END_VAR
(* ====================================================================== *)
(* *)
(* ====================================================================== *)
IF NOT Enable THEN
	Valid := FALSE;
	Error := FALSE;			(* reset at falling edge of Execute - just ErrorID will be kept til next rising edge *)
	ErrorID := 0;
END_IF
IF ReadMode = ReadMode_Once THEN
	fbTrigger(CLK:= Enable);
	IF fbTrigger.Q AND NOT bStarted THEN
		Value := 0;
		bStarted := TRUE;
		Valid := FALSE;
		Error := FALSE;
		ErrorID := MC_ERROR_NO_ERROR;
	END_IF;
ELSE
	IF Enable AND NOT bStarted THEN
		bStarted := TRUE;
		Valid := FALSE;
		Error := FALSE;
		ErrorID := MC_ERROR_NO_ERROR;
	END_IF;
	IF NOT Enable AND NOT bStarted THEN
		Valid := FALSE;
		Error := FALSE;
		ErrorID := MC_ERROR_NO_ERROR;
	END_IF;
END_IF;

IF bStarted THEN
	nParatype := PARAMETERTYPE_LREAL;
	fbReadWriteParameter(Enable:= TRUE, ParameterNumber:= ParameterNumber, Mode:= READWRITEPARAMETERMODE_READ,
						ParameterType:=nParatype, Axis:= Axis, ValueLreal:= Value, ValueDword := dwValue, ValueBool := bValue);
	IF fbReadWriteParameter.Done THEN
		bStarted := FALSE;
		Valid := TRUE;
		fbReadWriteParameter(Enable:= FALSE, ParameterNumber:= ParameterNumber, Mode:= READWRITEPARAMETERMODE_READ,
						ParameterType:= nParatype , Axis:= Axis, ValueLreal:= Value, ValueDword := dwValue, ValueBool := bValue);
	END_IF;
	IF fbReadWriteParameter.Error THEN
		Value := 0;
		bStarted := FALSE;
		Valid := FALSE;
		Error := TRUE;
		ErrorID := fbReadWriteParameter.ErrorID;
		fbReadWriteParameter(Enable:= FALSE, ParameterNumber:= ParameterNumber, Mode:= READWRITEPARAMETERMODE_READ,
						ParameterType:= nParatype , Axis:= Axis, ValueLreal:= Value, ValueDword := dwValue, ValueBool := bValue);
	END_IF;
END_IF;

ADSbusy := fbReadWriteParameter.ADSbusy;
Busy := (Enable AND ReadMode<>ReadMode_Once) OR bStarted;
END_FUNCTION_BLOCK

(* POU MC_ExtSetPointGenDisable, ST *)
FUNCTION_BLOCK MC_ExtSetPointGenDisable
VAR_IN_OUT
	Axis	:	AXIS_REF;
END_VAR
VAR_INPUT
	Execute : BOOL;
END_VAR
VAR_OUTPUT
	Done : BOOL;
	Busy: BOOL;
	Error: BOOL;
	ErrorID: UDINT;
	Enabled: BOOL;
END_VAR
VAR
	LastExecutionResult	: 	_ST_FunctionBlockResults;
	iState				:	_E_TcMC_STATES := STATE_INITIALIZATION;
	ADSbusy			: 	BOOL;
	fbADSwrite			: 	ADSWRITE;
END_VAR
{library private}
VAR
	fbOnTrigger			: 	R_TRIG;
	TimerStateFeedback	:	TON;
END_VAR
fbOnTrigger(CLK:= Execute);
Enabled := F_AxisHasExtSetPointGen(Axis.NcToPlc.StateDWord);

CASE iState OF
STATE_INITIALIZATION: (* initial iState *)
	Busy := FALSE;
	IF NOT Execute THEN
		Done := FALSE;
		Error := FALSE;
		ErrorID := 0;
	END_IF
	IF fbOnTrigger.Q THEN
		Busy := TRUE;
		(* initialization *)
		Done := FALSE;
		Error := FALSE;
		ErrorID := 0;
		LastExecutionResult.Done := FALSE;
		LastExecutionResult.CommandAborted := FALSE;
		LastExecutionResult.Error := FALSE;
		LastExecutionResult.ErrorID := 0;
		TimerStateFeedback(IN:=FALSE);
		fbADSwrite(WRITE:=FALSE);

		fbADSwrite(	NETID:= TcMcGlobal.NCNETID_TCMC,
					PORT:=AMSPORT_R0_NCSAF,
					IDXGRP:= TcMcGlobal.Axis.Functions.IDXGRP + Axis.NcToPlc.AxisId,
					IDXOFFS:= TCMCGLOBAL.Axis.Functions.IDXOFFS.DISABLEEXTGEN,
					LEN:=0,
					SRCADDR:=0,
					WRITE:=TRUE ,
					TMOUT:= TcMcGlobal.tADSTimeOut);
		iState := STATE_ORDER;
	END_IF

STATE_ORDER:  (* wait until command is accepted *)
	fbADSwrite(WRITE:= TRUE);
	IF NOT fbADSwrite.BUSY THEN
		Error := fbADSwrite.ERR;
		ErrorID := fbADSwrite.ERRID;
		IF NOT Error THEN
			IF NOT F_AxisHasExtSetPointGen(Axis.NcToPlc.StateDWord) THEN
				Done := TRUE;
				Busy := FALSE;
				iState := STATE_INITIALIZATION;
			ELSE
				iState := STATE_RUNNING;
			END_IF
		ELSE
			Busy := FALSE;
			iState := STATE_INITIALIZATION;
		END_IF
		Axis.PlcToNc.PlcCycleControl := 0; (* disable PLC cycle control *)
		LastExecutionResult.Done := Done;
		LastExecutionResult.Error := Error;
		LastExecutionResult.ErrorID := ErrorID;
	END_IF

STATE_RUNNING: (* wait for feedback flag from StateDWord *)
	TimerStateFeedback(IN:=TRUE, PT:=t#50ms);
	IF NOT F_AxisHasExtSetPointGen(Axis.NcToPlc.StateDWord) THEN
		Done := TRUE;
		Busy := FALSE;
		LastExecutionResult.Done := Done;
		LastExecutionResult.Error := Error;
		LastExecutionResult.ErrorID := ErrorID;
		iState := STATE_INITIALIZATION;
	ELSIF TimerStateFeedback.Q THEN
		(* the status flag 'external set point generator enabled' does not turn to TRUE *)
		Done := FALSE;
		Busy := FALSE;
		Error := TRUE;
		ErrorID := MC_ERROR_STATE_FEEDBACK_TIMEOUT;
		LastExecutionResult.Done := Done;
		LastExecutionResult.Error := Error;
		LastExecutionResult.ErrorID := ErrorID;
		iState := STATE_INITIALIZATION;
	END_IF
END_CASE

ADSbusy := fbAdsWrite.BUSY;
END_FUNCTION_BLOCK

(* POU MC_ExtSetPointGenEnable, ST *)
FUNCTION_BLOCK MC_ExtSetPointGenEnable
VAR_IN_OUT
	Axis	:	AXIS_REF;
END_VAR
VAR_INPUT
	Execute : BOOL;
	Position : LREAL;
	PositionType : E_PositionType;
END_VAR
VAR_OUTPUT
	Done : BOOL;
	Busy: BOOL;
	Error: BOOL;
	ErrorID: UDINT;
	Enabled: BOOL;
END_VAR
VAR
	LastExecutionResult	: 	_ST_FunctionBlockResults;
	iState				:	_E_TcMC_STATES := STATE_INITIALIZATION;
	ADSbusy			: 	BOOL;
	sExtSetPointGen 		: 	_ST_TcNC_SetPos;
	fbADSwrite			: 	ADSWRITE;
END_VAR
{library private}
VAR
	fbOnTrigger			: 	R_TRIG;
	TimerStateFeedback	:	TON;
END_VAR
fbOnTrigger(CLK:= Execute);
Enabled := F_AxisHasExtSetPointGen(Axis.NcToPlc.StateDWord);

CASE iState OF
STATE_INITIALIZATION: (* initial iState *)
	Busy := FALSE;
	IF NOT Execute THEN
		Done := FALSE;
		Error := FALSE;
		ErrorID := 0;
	END_IF
	IF fbOnTrigger.Q THEN
		Busy := TRUE;
		(* initialization *)
		Done := FALSE;
		Error := FALSE;
		ErrorID := 0;
		LastExecutionResult.Done := FALSE;
		LastExecutionResult.CommandAborted := FALSE;
		LastExecutionResult.Error := FALSE;
		LastExecutionResult.ErrorID := 0;
		TimerStateFeedback(IN:=FALSE);
		fbADSwrite(WRITE:=FALSE);

		sExtSetPointGen.fNewPosIst:=Position;
		sExtSetPointGen.nPosIstType:=PositionType;
		fbADSwrite(	NETID:= TcMcGlobal.NCNETID_TCMC,
					PORT:=AMSPORT_R0_NCSAF,
					IDXGRP:= TcMcGlobal.Axis.Functions.IDXGRP + Axis.NcToPlc.AxisId,
					IDXOFFS:= TCMCGLOBAL.Axis.Functions.IDXOFFS.ENABLEEXTGEN,
					LEN:=SIZEOF(sExtSetPointGen),
					SRCADDR:=ADR(sExtSetPointGen),
					WRITE:=TRUE ,
					TMOUT:= TcMcGlobal.tADSTimeOut);
		iState := STATE_ORDER;
	END_IF

STATE_ORDER:  (* wait until command is accepted *)
	fbADSwrite(WRITE:= TRUE);
	IF NOT fbADSwrite.BUSY THEN
		Error := fbADSwrite.ERR;
		ErrorID := fbADSwrite.ERRID;
		IF NOT Error THEN
			IF F_AxisHasExtSetPointGen(Axis.NcToPlc.StateDWord) THEN
				Done := TRUE;
				Busy := FALSE;
				iState := STATE_INITIALIZATION;
			ELSE
				iState := STATE_RUNNING;
			END_IF
		ELSE
			Busy := FALSE;
			iState := STATE_INITIALIZATION;
		END_IF
		LastExecutionResult.Done := Done;
		LastExecutionResult.Error := Error;
		LastExecutionResult.ErrorID := ErrorID;
	END_IF

STATE_RUNNING: (* wait for feedback flag from StateDWord *)
	TimerStateFeedback(IN:=TRUE, PT:=t#50ms);
	IF F_AxisHasExtSetPointGen(Axis.NcToPlc.StateDWord) THEN
		Done := TRUE;
		Busy := FALSE;
		LastExecutionResult.Done := Done;
		LastExecutionResult.Error := Error;
		LastExecutionResult.ErrorID := ErrorID;
		iState := STATE_INITIALIZATION;
	ELSIF TimerStateFeedback.Q THEN
		(* the status flag 'external set point generator enabled' does not turn to TRUE *)
		Done := FALSE;
		Busy := FALSE;
		Error := TRUE;
		ErrorID := MC_ERROR_STATE_FEEDBACK_TIMEOUT;
		LastExecutionResult.Done := Done;
		LastExecutionResult.Error := Error;
		LastExecutionResult.ErrorID := ErrorID;
		iState := STATE_INITIALIZATION;
	END_IF
END_CASE

ADSbusy := fbAdsWrite.BUSY;
END_FUNCTION_BLOCK

(* POU MC_ExtSetPointGenFeed, ST *)
FUNCTION MC_ExtSetPointGenFeed : BOOL
VAR_IN_OUT
	Axis	:	AXIS_REF;
END_VAR
VAR_INPUT
	Position		: LREAL;
	Velocity		: LREAL;
	Acceleration	: LREAL;
	Direction 	: DINT;
END_VAR
VAR
	GetTaskIndex : GETCURTASKINDEX;
END_VAR
Axis.PlcToNc.ExtSetPos := Position;
Axis.PlcToNc.ExtSetVelo := Velocity;
Axis.PlcToNc.ExtSetAcc := Acceleration;
Axis.PlcToNc.ExtSetDirection := Direction;

GetTaskIndex();
Axis.PlcToNc.PlcCycleControl.0 := 1; (* activate PLC cycle information to NC *)
Axis.PlcToNc.PlcCycleControl.1 := SystemTaskInfoArr[ GetTaskIndex.index ].cycleTimeExceeded;
Axis.PlcToNc.PlcCycleCount := Axis.PlcToNc.PlcCycleCount + 1;
END_FUNCTION

(* POU MC_GearIn, ST *)
FUNCTION_BLOCK MC_GearIn
(*	This Function Block commands a ratio between the velocity of the slave and master axis. *)
VAR_IN_OUT
	Master			:	AXIS_REF;		(* B *)
	Slave			:	AXIS_REF;		(* B *)
END_VAR
VAR_INPUT
	Execute			:	BOOL;			(* B *)
(*	ContinuousUpdate :	BOOL; *)			(* E *)	(* not available *)
	RatioNumerator	:	LREAL			(* B *)	:= 1; (* changed from INT (PLCopen) to LREAL *)
	RatioDenominator	:	UINT			(* B *)	:= 1;
(*	MasterValueSource :	MC_SOURCE; *)	(* E *)	(* not available *)
	Acceleration		:	LREAL;			(* E *)
	Deceleration		:	LREAL;			(* E *)
	Jerk				:	LREAL;			(* E *)
	BufferMode		:	MC_BufferMode;	(* E *)
	Options			: 	ST_GearInOptions;(* V *)	(* optional parameters *)
END_VAR
VAR_OUTPUT
	InGear			:	BOOL;	(* B *)
	Busy			: 	BOOL;	(* E *)
	Active			: 	BOOL;	(* E *)
	CommandAborted	:	BOOL;	(* E *)
	Error			:	BOOL;	(* B *)
	ErrorID			:	UDINT;	(* E *)
END_VAR
VAR
	LastExecutionResult	: 	_ST_FunctionBlockResults;
	ADSbusy: BOOL;
	iState				:	_E_TcMC_STATES := STATE_INITIALIZATION;
	fbAdsWrite			:	ADSWRITE;
	sCouple				:	_ST_TcNC_CoupleSlave;
	fbOptGearInDyn		: 	MC_GearInDyn;
END_VAR
{library private}
VAR
	fbOnTrigger			:	R_TRIG;
	TimerStateFeedback	: 	TON;
END_VAR
fbOnTrigger(CLK:= Execute);

CASE iState OF
STATE_INITIALIZATION:	(* *)
	Busy := FALSE;
	IF NOT Execute THEN
		InGear := FALSE;
		CommandAborted := FALSE;
		Error := FALSE;			(* reset at falling edge of Execute *)
		ErrorID := 0;
	END_IF
	IF fbOnTrigger.Q THEN
		Busy := TRUE;
		(* initialize output values *)
		InGear 			:= FALSE;
		CommandAborted	:= FALSE;
		ErrorID := 0;
		Error := FALSE;
		LastExecutionResult.Done := FALSE;
		LastExecutionResult.CommandAborted := FALSE;
		LastExecutionResult.Error := FALSE;
		LastExecutionResult.ErrorID := 0;
		fbOptGearInDyn.Enable := FALSE;
		TimerStateFeedback(IN:=FALSE);

		IF RatioDenominator = 0 THEN
			Error := TRUE;
			ErrorID := MC_ERROR_PARAMETER_NOT_CORRECT;
		ELSIF BufferMode <> 0 THEN
			Error := TRUE;
			ErrorID := MC_ERROR_BUFFERMODE_NOT_SUPPORTED;
		ELSE
			CASE Options.SlaveType OF
				0, TCNC_SLAVETYPE_LINEAR :
					(* linear gear ratio coupling *)
					sCouple.nSlaveType 		:= INT_TO_UDINT(TCNC_SLAVETYPE_LINEAR); (* linear coupling *)
					sCouple.nMasterAxisId		:= Master.NcToPlc.AxisId;
					sCouple.nMasterSubIdx	:= 0;
					sCouple.nSlaveSubIdx		:= 0;
					sCouple.fCoupleParam1	:= RatioNumerator / RatioDenominator;
					sCouple.fCoupleParam2	:= 0;(* unused *)
					sCouple.fCoupleParam3	:= 0;(* unused *)
					sCouple.fCoupleParam4	:= 0;(* unused *)
		
					fbAdsWrite(	NETID:= TcMcGlobal.NCNETID_TCMC,
							PORT:= TcMcGlobal.NCPORT_TCMC_COUPLING,
							IDXGRP:=TcMcGlobal.Axis.Functions.IDXGRP+Slave.NcToPlc.AxisId,
							IDXOFFS:= TcMcGlobal.Axis.Functions.IDXOFFS.CPL,
							LEN:= SIZEOF(sCouple),
							SRCADDR:= ADR(sCouple),
							WRITE:= TRUE,
							TMOUT:= TcMcGlobal.tADSTimeOut);
					iState := STATE_ORDER;

				TCNC_SLAVETYPE_LINEAR_CYCLICCHANGES_RAMP,
				TCNC_SLAVETYPE_CONST_SURFACEVELO_RAMP :
					fbOptGearInDyn.Enable := TRUE;
					ActGearInDyn();
					iState := STATE_ORDER;
			ELSE
				Error := TRUE;	(* Optional mode not supported with this function block *)
				ErrorID := MC_ERROR_PARAMETER_NOT_CORRECT;
			END_CASE
		END_IF;
	END_IF;

STATE_ORDER:
	CASE Options.SlaveType OF
		0, TCNC_SLAVETYPE_LINEAR :
			fbAdsWrite();
			IF NOT fbAdsWrite.Busy THEN
				IF fbAdsWrite.Err THEN
					ErrorID := fbAdsWrite.ErrId;
					Error := TRUE;
					iState := STATE_INITIALIZATION;
				ELSE
					iState := STATE_RUNNING;
				END_IF
				fbAdsWrite(WRITE := FALSE);
			END_IF;

		(* optional modes to couple with dynamically changable gear ratio (just couple) *)
		TCNC_SLAVETYPE_LINEAR_CYCLICCHANGES_RAMP,
		TCNC_SLAVETYPE_CONST_SURFACEVELO_RAMP :
			ActGearInDyn();
			IF fbOptGearInDyn.InGear THEN
				InGear := TRUE;
				fbOptGearInDyn.Enable := FALSE;
				ActGearInDyn();
				iState := STATE_INITIALIZATION;
			ELSIF NOT fbOptGearInDyn.Busy THEN
				CommandAborted := fbOptGearInDyn.CommandAborted;
				Error := fbOptGearInDyn.Error;
				ErrorID := fbOptGearInDyn.ErrorID;
				fbOptGearInDyn.Enable := FALSE;
				iState := STATE_INITIALIZATION;
			END_IF
	ELSE
		Error := TRUE;	(* Optional mode not supported with this function block *)
		ErrorID := MC_ERROR_PARAMETER_NOT_CORRECT;
		iState := STATE_INITIALIZATION;
	END_CASE

STATE_RUNNING:  (* Return *)
	TimerStateFeedback(IN:=TRUE, PT:=t#50ms); (* 21.2.2006 KSt *)
	IF  (Slave.NcToPlc.CoupleState = 2) OR (Slave.NcToPlc.CoupleState = 3) THEN
		(* axis successfully coupled *)
		InGear := TRUE;
		iState := STATE_INITIALIZATION;
	ELSIF TimerStateFeedback.Q THEN
		(* 	nCoupleState does not respond 'coupled' - the reason may be
			a MC_GearOut command which aborted the GearIn command *)
		CommandAborted := TRUE;
		iState := STATE_INITIALIZATION;
	END_IF;

ELSE  (* CASE : Unknown program state *)
	Error := TRUE;
	ErrorID := 16#FFFFFFFF;
	iState:= STATE_INITIALIZATION;
END_CASE

ADSbusy := fbAdsWrite.BUSY;
IF iState=STATE_INITIALIZATION THEN
	(* reset Busy immediately  when sequence ends *)
	IF Busy THEN
		LastExecutionResult.Done := InGear;
		LastExecutionResult.CommandAborted := CommandAborted;
		LastExecutionResult.Error := Error;
		LastExecutionResult.ErrorID := ErrorID;
	END_IF
	Busy := FALSE;
END_IF

Active := Busy;
END_FUNCTION_BLOCK
ACTION ActGearInDyn:
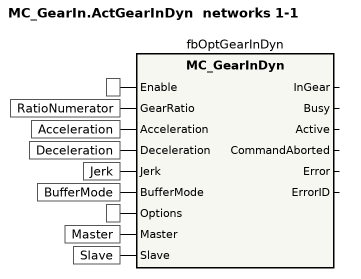
_FBD_ (* Function Block Diagram *)
NETWORK 1
	fbOptGearInDyn:MC_GearInDyn(Enable: , GearRatio: RatioNumerator, Acceleration: Acceleration, Deceleration: Deceleration, Jerk: Jerk, BufferMode: BufferMode, Options: , Master: Master, Slave: Slave)
_END_FBD_
END_ACTION
ACTION WriteGearRatio:
	(* action can be called from external in case of coupling modes with dynamically changable gear ratio *)
	IF RatioDenominator = 0 THEN
		Slave.PlcToNc.AxisModeLReal := RatioNumerator;
	ELSE
		Slave.PlcToNc.AxisModeLReal := RatioNumerator / RatioDenominator;
	END_IF
END_ACTION

(* POU MC_GearInDyn, ST *)
FUNCTION_BLOCK MC_GearInDyn
(*	MC_GearInDyn couples a slave axis to a master axis
 *	using a floating point gear ratio. The gear ratio can be 
 *	dynamically modified every PLC cycle as long as the 
 *	Execute input is TRUE.
 *	The acceleration input specifies the maximum slave
 *	acceleration in case of high gear ratio changes.
 *)
VAR_IN_OUT
	Master			:	AXIS_REF;
	Slave			:	AXIS_REF;
END_VAR
VAR_INPUT
	Enable			:	BOOL;
	GearRatio		:	LREAL := 1.0;
	Acceleration		:	LREAL;
	Deceleration		:	LREAL;	(* not used *)
	Jerk				:	LREAL;	(* not used *)
	BufferMode		:	MC_BufferMode;	(* E *)
	Options			: 	ST_GearInDynOptions;	(* V *)	(* optional parameters *)
END_VAR
VAR_OUTPUT
	InGear				:	BOOL;
	Busy				: 	BOOL;
	Active				: 	BOOL;
	CommandAborted		:	BOOL;
	Error				:	BOOL;
	ErrorID				:	UDINT;
END_VAR
VAR
	LastExecutionResult: 	_ST_FunctionBlockResults;
	ADSbusy: BOOL;
	iState			:	_E_TcMC_STATES := STATE_INITIALIZATION;
	iSubState		: 	INT;
	fbAdsWrite		:	ADSWRITE;
	fbAdsRead		:	ADSREAD;
	sCouple			:	_ST_TcNC_CoupleSlave;
	v_max			: 	LREAL;
	pa_limit			: 	LREAL;
	WasInGear: BOOL;
END_VAR
{library private}
VAR
	iAcceleration		: 	LREAL;
	TimerStateFeedback: TON;
END_VAR
CASE iState OF
	STATE_INITIALIZATION:	(* *)
		Busy := FALSE;
		Active := FALSE;
		IF Enable THEN
			Busy := TRUE;
			Active := TRUE;
			fbAdsRead(READ:=FALSE);
			fbAdsWrite(WRITE:=FALSE);
			(* initialize output values *)
			iAcceleration := Acceleration;
			ErrorID := 0;
			Error := FALSE;
			LastExecutionResult.Done := FALSE;
			LastExecutionResult.CommandAborted := FALSE;
			LastExecutionResult.Error := FALSE;
			LastExecutionResult.ErrorID := 0;
			TimerStateFeedback(IN:=FALSE);
			WasInGear := FALSE;
			iSubState := 0;

			IF BufferMode <> 0 THEN
				Error := TRUE;
				ErrorID := MC_ERROR_BUFFERMODE_NOT_SUPPORTED;
			ELSE
				InGear := F_AxisIsCoupled(Slave.NcToPlc.CoupleState) ;
				istate := SEL( InGear, STATE_ORDER, STATE_RUNNING);
			END_IF
		ELSE
			Error := FALSE;	(* reset at falling edge of Execute *)
			ErrorID := 0;
			CommandAborted := FALSE;
			InGear := FALSE;
		END_IF

	STATE_ORDER :
		Slave.PlcToNc.AxisModeLReal := GearRatio; (* 2008-06-02 KSt *)

		CASE iSubState OF
			0 :	(* read maximum master velocity *)
				fbAdsRead(	NETID:= TcMcGlobal.NCNETID_TCMC,
						PORT:= TcMcGlobal.NCPORT_TCMC,
						IDXGRP:=TcMcGlobal.Axis.Parameter.IDXGRP+Master.NcToPlc.AxisId,
						IDXOFFS:= TcMcGlobal.Axis.Parameter.IDXOFFS.VELOMAXIMUM,
						LEN:= SIZEOF(v_max),
						DESTADDR:= ADR(v_max),
						READ:= TRUE,
						TMOUT:= TcMcGlobal.tADSTimeOut);
				IF NOT fbAdsRead.Busy THEN
					Error := fbAdsRead.ERR;
					ErrorID := fbAdsRead.ERRID;
					fbAdsRead(READ:=FALSE);
					IF Error THEN
						iState := STATE_INITIALIZATION;
					ELSE
						iSubState := SEL(iAcceleration=0, iSubState + 2, iSubState + 1 );
					END_IF
				END_IF;

			1 :	(* read slave default acceleration *)
				fbAdsRead(	NETID:=TcMcGlobal.NCNETID_TCMC,
						PORT:= TcMcGlobal.NCPORT_TCMC,
						IDXGRP:=TcMcGlobal.Axis.Parameter.IDXGRP+Slave.NcToPlc.AxisId,
						IDXOFFS:= TcMcGlobal.Axis.Parameter.IDXOFFS.ACC,
						LEN:= SIZEOF(iAcceleration),
						DESTADDR:= ADR(iAcceleration),
						READ:= TRUE,
						TMOUT:= TcMcGlobal.tADSTimeOut);
				IF NOT fbAdsRead.Busy THEN
					Error := fbAdsRead.ERR;
					ErrorID := fbAdsRead.ERRID;
					fbAdsRead(READ:=FALSE);
					IF Error THEN
						iState := STATE_INITIALIZATION;
					ELSE
						iSubState := iSubState + 1;
					END_IF
				END_IF;

			2 : (* couple with dynamic gear ratio *)
				(* 	pa entspricht indirekt, naemlich bezogen auf eine maximale
					Mastergeschwindigkeit, einer maximal erlaubten 
					Beschleunigung (pa = aSlaveMax / vMasterMax ). 
					Der Begrenzungsparameter pa entspricht dabei dem 
					Kehrwert der Hochlaufzeit tH = 1 / pa . 
				*)
				IF iAcceleration > 0 AND v_max > 0 THEN
					pa_limit := iAcceleration / v_max;
				ELSE
					pa_limit := 1;
				END_IF

				sCouple.nSlaveType 	:= INT_TO_UDINT( SEL( Options.CCVmode,
					TCNC_SLAVETYPE_LINEAR_CYCLICCHANGES_RAMP,
					TCNC_SLAVETYPE_CONST_SURFACEVELO_RAMP) );
				sCouple.nMasterAxisId	:= Master.NcToPlc.AxisId;
				sCouple.nMasterSubIdx	:= 0;
				sCouple.nSlaveSubIdx		:= 0;
				sCouple.fCoupleParam1	:= pa_limit;
				sCouple.fCoupleParam2	:= 0;(* unused *)
				sCouple.fCoupleParam3	:= 0;(* unused *)
				sCouple.fCoupleParam4	:= 0;(* unused *)

				(* Slave.PlcToNc.AxisModeLReal := GearRatio;*) (* 2008-06-02 KSt *)

				fbAdsWrite(	NETID:= TcMcGlobal.NCNETID_TCMC,
						PORT:= TcMcGlobal.NCPORT_TCMC_COUPLING,
						IDXGRP:=TcMcGlobal.Axis.Functions.IDXGRP+Slave.NcToPlc.AxisId,
						IDXOFFS:= TcMcGlobal.Axis.Functions.IDXOFFS.CPL,
						LEN:= SIZEOF(sCouple),
						SRCADDR:= ADR(sCouple),
						WRITE:= TRUE,
						TMOUT:= TcMcGlobal.tADSTimeOut);
				IF NOT fbAdsWrite.Busy THEN
					Error := fbAdsWrite.ERR;
					ErrorID := fbAdsWrite.ERRID;
					fbAdsWrite(WRITE:=FALSE);
					IF Error THEN
						iState := STATE_INITIALIZATION;
					ELSE
						InGear := F_AxisIsCoupled(Slave.NcToPlc.CoupleState);
						iState := STATE_RUNNING;
					END_IF
				END_IF
		END_CASE

	STATE_RUNNING:  (* cyclic change of the gear ratio until decoupled or until Execute=FALSE *)
		TimerStateFeedback(IN:=TRUE, PT:=t#50ms); (* 5.7.2006 KSt *)
		Slave.PlcToNc.AxisModeLReal := GearRatio;
		InGear := F_AxisIsCoupled(Slave.NcToPlc.CoupleState) ;
		IF InGear THEN
			WasInGear := TRUE; (* feedback seen, 5.7.2006 KSt *)
		END_IF
		IF (NOT Enable OR NOT InGear) AND (WasInGear OR TimerStateFeedback.Q) THEN (* 5.7.2006 KSt *)
			(* Slave.PlcToNc.AxisModeLReal := 0;*) (* stop when still in gear but not enabled *) (* keep latest gear ratio - 2009-02-19 KSt *)
			CommandAborted := NOT InGear;
			iState := STATE_INITIALIZATION;
		END_IF;

	ELSE  (* CASE : Unknown program state *)
		Error := TRUE;
		ErrorID := 16#FFFFFFFF;
		iState:= STATE_INITIALIZATION;
END_CASE

ADSbusy := fbAdsWrite.BUSY OR fbAdsRead.BUSY;
IF iState=STATE_INITIALIZATION THEN
	(* reset Busy immediately  when sequence ends *)
	IF Busy THEN
		LastExecutionResult.Done := InGear;
		LastExecutionResult.CommandAborted := CommandAborted;
		LastExecutionResult.Error := Error;
		LastExecutionResult.ErrorID := ErrorID;
	END_IF
	Busy := FALSE;
	Active := FALSE;
END_IF
END_FUNCTION_BLOCK

(* POU MC_GearInMultiMaster, ST *)
FUNCTION_BLOCK MC_GearInMultiMaster
(*	MC_GearInDyn couples a slave axis to a master axis
 *	using a floating point gear ratio. The gear ratio can be 
 *	dynamically modified every PLC cycle as long as the 
 *	Execute input is TRUE.
 *	The acceleration input specifies the maximum slave
 *	acceleration in case of high gear ratio changes.
 *)
VAR_IN_OUT
	Master1			:	AXIS_REF;
	Master2			:	AXIS_REF;
	Master3			:	AXIS_REF;
	Master4			:	AXIS_REF;
	Slave			:	AXIS_REF;
END_VAR
VAR_INPUT
	Enable			:	BOOL;
	GearRatio1		:	LREAL := 1.0;
	GearRatio2		:	LREAL := 1.0;
	GearRatio3		:	LREAL := 1.0;
	GearRatio4		:	LREAL := 1.0;
	Acceleration		:	LREAL;
	Deceleration		:	LREAL;	(* just used in version 2 mode (AdvancedSlaveDynamics) *)
	Jerk				:	LREAL;	(* just used in version 2 mode (AdvancedSlaveDynamics) *)
	BufferMode		:	MC_BufferMode;	(* E *)
	Options			: 	ST_GearInMultiMasterOptions;	(* V *)	(* optional parameters *)
END_VAR
VAR_OUTPUT
	InGear				:	BOOL;
	Busy				: 	BOOL;
	Active				: 	BOOL;
	CommandAborted		:	BOOL;
	Error				:	BOOL;
	ErrorID				:	UDINT;
END_VAR
VAR
	InGear2				:	BOOL; (* new internal feedback flag 2015-10-19 FAp *)
	ADSbusy			: 	BOOL;
	iState				:	_E_TcMC_STATES := STATE_INITIALIZATION;
	fbAdsWrite			:	ADSWRITE;
	sCouple				:	_ST_TcNC_CoupleSlaveMultiMaster;
	sCoupleV2			:	_ST_TcNC_CoupleSlaveMultiMaster2;
	LastExecutionResult	: 	_ST_FunctionBlockResults;
	IsCoupled			: 	BOOL;
END_VAR
{library private}
VAR
	TimerStateFeedback	: 	TON;
	iAdvancedSlaveDynamics:	BOOL;
	iAcceleration			: 	LREAL;
	iDeceleration			:	LREAL;	(* just used in version 2 mode *)
	iJerk				:	LREAL;	(* just used in version 2 mode *)
	WasInGear			:	 BOOL;
	ParameterChanged	:	 BOOL;
	i					:	UDINT; (* runtime optimization 2015-10-19 FAp *)
	InGear2Cnt			:	UDINT; (* runtime optimization 2015-10-19 FAp *)
	LastNcCycleCounter	:	UDINT; (* runtime optimization 2015-10-19 FAp *)
END_VAR
IF Enable AND NOT Busy THEN
	(* AdvancedSlaveDynamics can only be changed when triggered *)
	iAdvancedSlaveDynamics := Options.AdvancedSlaveDynamics;
END_IF

IF iAdvancedSlaveDynamics THEN
	ActGearInMultiMasterV2();	(* new version V2 - 2011-09-07 KSt *)
ELSE
	ActGearInMultiMasterV1();	(* classic version V1 *)
END_IF
END_FUNCTION_BLOCK
ACTION ActGearInMultiMasterV1:
(*
 *	CLASSIC   MC_GearInMultimaster 
 *)
CASE iState OF
	STATE_INITIALIZATION:	(* *)
		Busy := FALSE;
		Active := FALSE;
		IF Enable THEN
			Busy := TRUE;
			Active := TRUE;
			fbAdsWrite(WRITE:=FALSE);
			(* initialize output values *)
			iAcceleration := Acceleration;
			ErrorID := 0;
			Error := FALSE;
			LastExecutionResult.Done := FALSE;
			LastExecutionResult.CommandAborted := FALSE;
			LastExecutionResult.Error := FALSE;
			LastExecutionResult.ErrorID := 0;
			TimerStateFeedback(IN:=FALSE);
			WasInGear := FALSE;

			IF BufferMode <> 0 THEN
				Error := TRUE;
				ErrorID := MC_ERROR_BUFFERMODE_NOT_SUPPORTED;
			ELSE
				InGear := F_AxisIsCoupled(Slave.NcToPlc.CoupleState) ;
				istate := SEL( InGear, STATE_ORDER, STATE_RUNNING);
			END_IF

		ELSE
			Error := FALSE;	(* reset when Enable is FALSE *)
			ErrorID := 0;
			CommandAborted := FALSE;
			InGear := FALSE;
		END_IF

	STATE_ORDER :
			(* couple with dynamic gear ratio *)
			sCouple.nSlaveType := INT_TO_UDINT(TCNC_SLAVETYPE_LINEAR_MULTIMASTER);
			sCouple.nMasterSubIdx	:= 0;
			sCouple.nSlaveSubIdx		:= 0;
(*			sCouple.fCoupleParam1	:= iAcceleration;*)
			sCouple.nMasterAxisId := Master1.NcToPlc.AxisId;
			sCouple.nMasterID2 := Master2.NcToPlc.AxisId;
			sCouple.nMasterID3 := Master3.NcToPlc.AxisId;
			sCouple.nMasterID4 := Master4.NcToPlc.AxisId;
			sCouple.fSlaveAcceleration := iAcceleration;
(* 			sCouple.nCheckAndOpMode := ? *)

			(* cyclic data *)
			Slave.PlcToNc.GearRatio1 := GearRatio1;
			Slave.PlcToNc.GearRatio2 := GearRatio2;
			Slave.PlcToNc.GearRatio3 := GearRatio3;
			Slave.PlcToNc.GearRatio4 := GearRatio4;

			fbAdsWrite(	NETID:= TcMcGlobal.NCNETID_TCMC,
					PORT:= TcMcGlobal.NCPORT_TCMC_COUPLING,
					IDXGRP:=TcMcGlobal.Axis.Functions.IDXGRP+Slave.NcToPlc.AxisId,
					IDXOFFS:= TcMcGlobal.Axis.Functions.IDXOFFS.CPL,
					LEN:= SIZEOF(sCouple),
					SRCADDR:= ADR(sCouple),
					WRITE:= TRUE,
					TMOUT:= TcMcGlobal.tADSTimeOut);
			IF NOT fbAdsWrite.Busy THEN
				Error := fbAdsWrite.ERR;
				ErrorID := fbAdsWrite.ERRID;
				fbAdsWrite(WRITE:=FALSE);
				IF Error THEN
					iState := STATE_INITIALIZATION;
				ELSE
					InGear := F_AxisIsCoupled(Slave.NcToPlc.CoupleState);
					iState := STATE_RUNNING;
				END_IF
			END_IF

	STATE_RUNNING:  (* cyclic change of the gear ratio until decoupled or until Execute=FALSE *)
		TimerStateFeedback(IN:=TRUE, PT:=t#50ms); (* 5.7.2006 KSt *)
		Slave.PlcToNc.GearRatio1 := GearRatio1;
		Slave.PlcToNc.GearRatio2 := GearRatio2;
		Slave.PlcToNc.GearRatio3 := GearRatio3;
		Slave.PlcToNc.GearRatio4 := GearRatio4;
		InGear := F_AxisIsCoupled(Slave.NcToPlc.CoupleState) ;
		IF InGear THEN
			WasInGear := TRUE; (* feedback seen, 5.7.2006 KSt *)
		END_IF
		IF (NOT Enable OR NOT InGear) AND (WasInGear OR TimerStateFeedback.Q) THEN (* 5.7.2006 KSt *)
(*  keep latest gear ratio - 2008-02-19 KSt *)
			(* stop when still in gear but not enabled *)
(*			Slave.PlcToNc.GearRatio1 := 0;
			Slave.PlcToNc.GearRatio2 := 0;
			Slave.PlcToNc.GearRatio3 := 0;
			Slave.PlcToNc.GearRatio4 := 0;
*)
			CommandAborted := NOT InGear;
			iState := STATE_INITIALIZATION;
		END_IF;

	ELSE  (* CASE : Unknown program state *)
		Error := TRUE;
		ErrorID := 16#FFFFFFFF;
		iState:= STATE_INITIALIZATION;
END_CASE

ADSbusy := fbAdsWrite.BUSY;
IF iState=STATE_INITIALIZATION THEN
	(* reset Busy immediately  when sequence ends *)
	IF Busy THEN
		LastExecutionResult.Done := InGear;
		LastExecutionResult.CommandAborted := CommandAborted;
		LastExecutionResult.Error := Error;
		LastExecutionResult.ErrorID := ErrorID;
	END_IF
	Busy := FALSE;
	Active := FALSE;
END_IF
END_ACTION
ACTION ActGearInMultiMasterV2:
(*
 *	EXTENDED   MC_GearInMultimaster Version 2
 *	2011-09-07 KSt 
 *)
FOR i := 1 TO 2 DO  (* runtime optimization 2015-10-19 FAp *)
	CASE iState OF
		STATE_INITIALIZATION:	(* *)
			Busy := FALSE;
			Active := FALSE;
			IF Enable THEN
				Busy := TRUE;
				Active := TRUE;
				fbAdsWrite(WRITE:=FALSE);
				(* initialize output values *)
				iAcceleration := Acceleration;
				iDeceleration := Deceleration;
				iJerk := Jerk;
				ErrorID := 0;
				Error := FALSE;
				LastExecutionResult.Done := FALSE;
				LastExecutionResult.CommandAborted := FALSE;
				LastExecutionResult.Error := FALSE;
				LastExecutionResult.ErrorID := 0;
				TimerStateFeedback(IN:=FALSE);
				WasInGear := FALSE;
	
				IF BufferMode <> 0 THEN
					Error := TRUE;
					ErrorID := MC_ERROR_BUFFERMODE_NOT_SUPPORTED;
					EXIT;
				ELSE
					IsCoupled := F_AxisIsCoupled(Slave.NcToPlc.CoupleState) ;
					istate := SEL( IsCoupled, STATE_ORDER, STATE_RUNNING);
				END_IF
			ELSE
				Error := FALSE;	(* reset when Enable is FALSE *)
				ErrorID := 0;
				CommandAborted := FALSE;
				InGear := FALSE;
				InGear2 := FALSE; (* new internal feedback flag 2015-10-19 FAp *)
				EXIT;
			END_IF

		STATE_ORDER :
			IsCoupled := F_AxisIsCoupled(Slave.NcToPlc.CoupleState) ;
			InGear := Slave.NcToPlc.AxisState=INT_TO_DWORD(TCNC_PHASE_SYNCHRONOUS);
			InGear2 := FALSE;

			(* couple with dynamic gear ratio *)
			sCoupleV2.nSlaveType := INT_TO_UDINT(TCNC_SLAVETYPE_LINEAR_MULTIMASTER);
			sCoupleV2.nMasterSubIdx	:= 0;
			sCoupleV2.nSlaveSubIdx	:= 0;
			IF NOT IsCoupled THEN
				sCoupleV2.nMasterAxisId := Master1.NcToPlc.AxisId;
				sCoupleV2.nMasterID2 := Master2.NcToPlc.AxisId;
				sCoupleV2.nMasterID3 := Master3.NcToPlc.AxisId;
				sCoupleV2.nMasterID4 := Master4.NcToPlc.AxisId;
			END_IF
			sCoupleV2.fSlaveMaxVelo := 0;	(* use axis default *)
			sCoupleV2.fSlaveMaxAcc := iAcceleration;
			sCoupleV2.fSlaveMaxDec := iDeceleration;
			sCoupleV2.fSlaveMaxJerk := iJerk;
			sCoupleV2.nCheckAndOpMode.0 := Options.VelocitySynchronizationOnly;	(* set bit 0 in bit array *)

			(* cyclic data *)
			Slave.PlcToNc.GearRatio1 := GearRatio1;
			Slave.PlcToNc.GearRatio2 := GearRatio2;
			Slave.PlcToNc.GearRatio3 := GearRatio3;
			Slave.PlcToNc.GearRatio4 := GearRatio4;

			fbAdsWrite(	NETID:= TcMcGlobal.NCNETID_TCMC,
					PORT:= TcMcGlobal.NCPORT_TCMC_COUPLING,
					IDXGRP:=TcMcGlobal.Axis.Functions.IDXGRP+Slave.NcToPlc.AxisId,
					IDXOFFS:= TcMcGlobal.Axis.Functions.IDXOFFS.CPL,
					LEN:= SIZEOF(sCoupleV2),
					SRCADDR:= ADR(sCoupleV2),
					WRITE:= TRUE,
					TMOUT:= TcMcGlobal.tADSTimeOut);
			IF NOT fbAdsWrite.Busy THEN
				Error := fbAdsWrite.ERR;
				ErrorID := fbAdsWrite.ERRID;
				fbAdsWrite(WRITE:=FALSE);
				IF Error THEN
					iState := STATE_INITIALIZATION;
				ELSE
					InGear2Cnt := 1;
					LastNcCycleCounter := DWORD_TO_BYTE(SHR(Slave.NcToPlc.OpModeDWord, 24));
					iState := STATE_RUNNING;
				END_IF
			ELSE
				EXIT;
			END_IF

		STATE_RUNNING:  (* cyclic change of the gear ratio until decoupled or until Execute=FALSE *)
			TimerStateFeedback(IN:=TRUE, PT:=t#50ms); (* 5.7.2006 KSt *)

			(* new internal feedback flag 2015-10-19 FAp *)
			IF (Slave.PlcToNc.GearRatio1 <> GearRatio1)
			  OR (Slave.PlcToNc.GearRatio2 <> GearRatio2)
			  OR (Slave.PlcToNc.GearRatio3 <> GearRatio3)
			  OR (Slave.PlcToNc.GearRatio4 <> GearRatio4) THEN
				InGear2 := FALSE;
				InGear2Cnt := 0;
				LastNcCycleCounter := DWORD_TO_BYTE(SHR(Slave.NcToPlc.OpModeDWord, 24));
			END_IF

			Slave.PlcToNc.GearRatio1 := GearRatio1;
			Slave.PlcToNc.GearRatio2 := GearRatio2;
			Slave.PlcToNc.GearRatio3 := GearRatio3;
			Slave.PlcToNc.GearRatio4 := GearRatio4;
			IsCoupled := F_AxisIsCoupled(Slave.NcToPlc.CoupleState) ;
			InGear := Slave.NcToPlc.AxisState=INT_TO_DWORD(TCNC_PHASE_SYNCHRONOUS);

			(* new internal feedback flag 2015-10-19 FAp *)
			IF _F_NcCycleCounterUpdated(LastNcCycleCounter, Slave) AND InGear2Cnt < 2 THEN
				InGear2Cnt := InGear2Cnt + 1;
				LastNcCycleCounter := DWORD_TO_BYTE(SHR(Slave.NcToPlc.OpModeDWord, 24));
			END_IF	

			(* new internal feedback flag 2015-10-19 FAp *)
			IF InGear2Cnt >= 2 OR InGear2 THEN
				InGear2 := Slave.NcToPlc.AxisState=INT_TO_DWORD(TCNC_PHASE_SYNCHRONOUS);
			END_IF

			IF IsCoupled THEN
				WasInGear := TRUE; (* feedback seen, 5.7.2006 KSt *)
			END_IF
			IF (NOT Enable OR NOT IsCoupled) AND (WasInGear OR TimerStateFeedback.Q) THEN (* 5.7.2006 KSt *)
				CommandAborted := NOT IsCoupled;
				iState := STATE_INITIALIZATION;
			ELSE
				ParameterChanged :=
					(Acceleration <> iAcceleration) OR
					(Deceleration <> iDeceleration) OR
					(Jerk <> iJerk);
				IF ParameterChanged THEN
					iAcceleration := Acceleration;
					iDeceleration := Deceleration;
					iJerk := Jerk;
					istate := STATE_ORDER;
				ELSE
					EXIT;
				END_IF
			END_IF;
	
		ELSE  (* CASE : Unknown program state *)
			Error := TRUE;
			ErrorID := 16#FFFFFFFF;
			iState:= STATE_INITIALIZATION;
	END_CASE
END_FOR

ADSbusy := fbAdsWrite.BUSY;
IF iState=STATE_INITIALIZATION THEN
	(* reset Busy immediately  when sequence ends *)
	IF Busy THEN
		LastExecutionResult.Done := InGear;
		LastExecutionResult.CommandAborted := CommandAborted;
		LastExecutionResult.Error := Error;
		LastExecutionResult.ErrorID := ErrorID;
	END_IF
	Busy := FALSE;
	Active := FALSE;
END_IF
END_ACTION

(* POU MC_GearOut, ST *)
FUNCTION_BLOCK MC_GearOut
(*	This Function Block disengages the Slave axis from the Master axis.
	Notes:
	It is assumed that this command is followed by another command, for instance 
	MC_Stop, MC_GearIn, or any other command. If there is no new command, the 
	default condition should be: maintain last velocity.
 *)
VAR_IN_OUT
	Slave			:	AXIS_REF;	(* B *)
END_VAR
VAR_INPUT
	Execute			:	BOOL;		(* B *)
	Options			: 	ST_GearOutOptions;	(* V *)	(* optional parameters *)
END_VAR
VAR_OUTPUT
	Done			:	BOOL;		(* B *)
	Busy			: 	BOOL;		(* E *)
	Error			:	BOOL;		(* B *)
	ErrorID			:	UDINT;		(* E *)
END_VAR
VAR
	LastExecutionResult: 	_ST_FunctionBlockResults;
	ADSbusy		: 	BOOL;
	iState			:	_E_TcMC_STATES := STATE_INITIALIZATION;
	fbAdsWrite		:	ADSWRITE;
END_VAR
{library private}
VAR
	fbOnTrigger		:	R_TRIG;
	TimerStateFeedback: TON;
END_VAR
 fbOnTrigger(CLK:= Execute);

CASE iState OF
	STATE_INITIALIZATION:	(* *)
		Busy := FALSE;
		IF NOT Execute THEN
			Done := FALSE;
			Error := FALSE;			(* reset at falling edge of Execute *)
			ErrorID := 0;
		END_IF
	    	IF fbOnTrigger.Q THEN
			(* initialize output values *)
	    		Busy := TRUE;
			Done := FALSE;
			ErrorID := 0;
			Error := FALSE;
			LastExecutionResult.Done := FALSE;
			LastExecutionResult.CommandAborted := FALSE;
			LastExecutionResult.Error := FALSE;
			LastExecutionResult.ErrorID := 0;
			TimerStateFeedback(IN:=FALSE);
			fbAdsWrite(WRITE := FALSE);

			fbAdsWrite(	NETID:=TcMcGlobal.NCNETID_TCMC,
						PORT:= TcMcGlobal.NCPORT_TCMC_COUPLING, (* 12.7.2006 KSt *)
						IDXGRP:=TcMcGlobal.Axis.Functions.IDXGRP+Slave.NcToPlc.AxisId,
						IDXOFFS:= TcMcGlobal.Axis.Functions.IDXOFFS.DECPL,
						LEN:= 0,
						SRCADDR:= 0,
						WRITE:= TRUE,
						TMOUT:= TcMcGlobal.tADSTimeOut);

			iState := STATE_ORDER;
		END_IF;

	STATE_ORDER:
		fbAdsWrite();
		IF NOT fbAdsWrite.BUSY THEN
			IF fbAdsWrite.Err THEN
				Error := TRUE;
				ErrorID := fbAdsWrite.ErrId;
				fbAdsWrite(WRITE := FALSE);
				iState := STATE_INITIALIZATION;
			ELSE
				IF  (Slave.NcToPlc.CoupleState < 2) THEN
					(* axis successfully decoupled *)
					Done := TRUE;
					iState := STATE_INITIALIZATION;
				ELSE (* wait for Nc2Plc feedback *)
					(* Done := TRUE; *)					 (* removed 2012-12-22 KSt *)
					(* iState := STATE_INITIALIZATION; *)	 (* removed 2012-12-22 KSt *)
					iState := STATE_RUNNING;			 (* added 2012-12-22 KSt *)
				END_IF
				fbAdsWrite(WRITE := FALSE);
			END_IF;
		END_IF;

	STATE_RUNNING:  (* waiting for Nc2Plc feedback - added 2012-12-22 KSt *)
		TimerStateFeedback(IN:=TRUE, PT:=t#50ms);
		IF  (Slave.NcToPlc.CoupleState < 2) THEN
			(* axis successfully decoupled *)
			Done := TRUE;
			iState := STATE_INITIALIZATION;
		ELSIF TimerStateFeedback.Q THEN
			(* 	nCoupleState does not respond 'not coupled' 	*)
			Error := TRUE;
			ErrorID := MC_ERROR_STATE_FEEDBACK_TIMEOUT;
			iState := STATE_INITIALIZATION;
		END_IF;

	ELSE  (* CASE : Unknown program state *)
		Error := TRUE;
		ErrorID := 16#FFFFFFFF;
		iState:= STATE_INITIALIZATION;
END_CASE

ADSbusy := fbAdsWrite.BUSY;

IF iState=STATE_INITIALIZATION THEN
	(* reset Busy immediately  when sequence ends *)
	IF Busy THEN
		LastExecutionResult.Done := Done;
		LastExecutionResult.Error := Error;
		LastExecutionResult.ErrorID := ErrorID;
	END_IF
	Busy := FALSE;
END_IF
END_FUNCTION_BLOCK

(* POU MC_Home, ST *)
FUNCTION_BLOCK MC_Home
(*
	Function block defined by PLCopen Part 1 - Function blocks for motion control

	This Function Block commands the axis to perform the «search home» sequence.
	The details of this sequence can be set by the axis’ parameters. 
	The 'Position' input is used to set the absolute position when reference signal 
	is detected. This Function Bock completes at 'StandStill'.
*)
VAR_IN_OUT
	Axis				:	AXIS_REF;	(* B *)
END_VAR
VAR_INPUT
	Execute			:	BOOL;	(* B *)
	Position			:	LREAL	(* B *) := DEFAULT_HOME_POSITION;
	HomingMode		: 	MC_HomingMode;	(* V *)
	BufferMode		:	MC_BufferMode;		(* E *)
	Options			: 	ST_HomingOptions;	(* V *)	(* Beckhoff proprietary input *)
	bCalibrationCam 	: 	BOOL;	(* V *)	(* Beckhoff proprietary input *)
END_VAR
VAR_OUTPUT
	Done			:	BOOL;	(* B *)
	Busy			: 	BOOL;	(* E *)
	Active			: 	BOOL;	(* E *)
	CommandAborted	:	BOOL;	(* E *)
	Error			:	BOOL;	(* B *)
	ErrorID			:	UDINT;	(* E *)
END_VAR
VAR
	LastExecutionResult: 	_ST_FunctionBlockResults;
	ADSbusy		: 	BOOL;
	iState			: 	_E_TcMC_STATES := STATE_INITIALIZATION;
	iSubState		: 	INT;
	fbAdsWriteCmd	: 	ADSWRITE;
	fbAdsWriteRefPos: 	ADSWRITE;
	fbAdsReadRefPos: 	ADSREAD;
	ReferenceFlagValue: UDINT;
	fbSetPosition: MC_SetPosition;
	NcHomePosition 	:	LREAL;
END_VAR
{library private}
VAR
	fbTrigger			:	R_TRIG;
	fbTimeOut		:	TON;
END_VAR
(*
	PlcOpen comment to MC_Home:
		HomingMode input ist Beckhoff-spezifisch (war in vorheriger Spezifikation mal vorhanden)
		BufferMode ist nicht implementiert.
*)

 fbTrigger(CLK:= Execute);

CASE iSubState OF
	0 :	(* init *)
		iState := STATE_INITIALIZATION;	(* *)
		Busy := FALSE;
		IF NOT Execute THEN
			Done := FALSE;
			CommandAborted := FALSE;
			Error := FALSE;			(* reset at falling edge of Execute *)
			ErrorID := 0;
		END_IF
	   	IF fbTrigger.Q THEN
			(* initialize output values *)
	   		Busy := TRUE;
			Done := FALSE;
			CommandAborted := FALSE;
			Error := FALSE;
			ErrorID := 0;
			fbAdsWriteCmd(WRITE:=FALSE);
			fbAdsWriteRefPos(WRITE:=FALSE);
			fbAdsReadRefPos(READ:=FALSE);
			fbTimeOut(IN:=FALSE);
			fbSetPosition(	Execute:= FALSE, Axis:=Axis);

			IF BufferMode <> 0 THEN
		   		Busy := FALSE;
				Error := TRUE;
				ErrorID := MC_ERROR_BUFFERMODE_NOT_SUPPORTED;
			ELSE
				CASE HomingMode OF
					MC_DefaultHoming :
						IF Position < DEFAULT_HOME_POSITION THEN
							iSubState := iSubState + 1;	(* write home position before homing *)
						ELSE
							iSubState := iSubState + 2; 	(* start homing *)
						END_IF
					MC_Direct :
						ReferenceFlagValue := 1;
						IF Position < DEFAULT_HOME_POSITION THEN
							fbSetPosition.Position := Position;
							iSubState := 10;	(* set position and reference flag *)
						ELSE
							iSubState := 9; 	(* read homing position and then set position and reference flag *)
						END_IF
					MC_ForceCalibration :
						ReferenceFlagValue := 1;
						iSubState := 11; (* set reference flag *)
					MC_ResetCalibration :
						ReferenceFlagValue := 0;
						iSubState := 11; (* set reference flag *)
				ELSE (* case *)
			   		Busy := FALSE;
					Error := TRUE;
					ErrorID := MC_ERROR_CALIBRATION_ERROR; (* homing mode not supported *)
				END_CASE
			END_IF
		END_IF

	1 :	(* write homing position *)
		fbAdsWriteRefPos(	NETID:= TcMcGlobal.NCNETID_TCMC,
							PORT:= TcMcGlobal.NCPORT_TCMC,
							IDXGRP:=TcMcGlobal.Axis.Parameter.IDXGRP+Axis.NcToPlc.AxisId,
							IDXOFFS:= TcMcGlobal.Axis.Parameter.IDXOFFS.REF_POS,
							LEN:= SIZEOF(Position),
							SRCADDR:= ADR(Position),
							WRITE:= TRUE,
							TMOUT:= TcMcGlobal.tADSTimeOut);
		IF NOT fbAdsWriteRefPos.Busy THEN
			IF fbAdsWriteRefPos.Err	THEN
				Error := fbAdsWriteRefPos.ERR;
				ErrorID := fbAdsWriteRefPos.ERRID;
				iSubState := 0;
			ELSE
				NcHomePosition := Position;
				iSubState := iSubState + 1; (* start homing *)
			END_IF
		END_IF

	2 :	(* start homing *)
		fbAdsWriteCmd(	NETID:= TcMcGlobal.NCNETID_TCMC,
						PORT:= TcMcGlobal.NCPORT_TCMC,
						IDXGRP:=TcMcGlobal.Axis.Functions.IDXGRP+Axis.NcToPlc.AxisId,
						IDXOFFS:= TcMcGlobal.Axis.Functions.IDXOFFS.CALIBR,
						LEN:= 0,
						SRCADDR:= 0,
						WRITE:= TRUE,
						TMOUT:= TcMcGlobal.tADSTimeOut);
		IF NOT fbAdsWriteCmd.Busy THEN
			IF fbAdsWriteCmd.ERR THEN
				Error := fbAdsWriteCmd.ERR;
				ErrorID := fbAdsWriteCmd.ERRID;
				iSubState := 0;
			ELSE
				fbTimeOut(IN:=TRUE, PT:=TcMcGlobal.tADSTimeOut);
				IF fbTimeOut.Q THEN
					(* calibration sequence did not start *)
					Error 	:= TRUE;
					ErrorID := MC_ERROR_CALIBRATION_ERROR; (* functional/calibration error *)
					iSubState := 0;
				END_IF;
				IF F_AxisIsCalibrating(StateDWord := Axis.NcToPlc.StateDWord) THEN
					(* calibration sequence started *)
					iState := STATE_RUNNING;
					iSubState := iSubState + 1; (* wait homing *)
				END_IF
			END_IF
		END_IF

	3 :	(* homing Busy *)
		(* wait for done in cyclic interface *)
		IF NOT F_AxisIsCalibrating(StateDWord := Axis.NcToPlc.StateDWord) THEN
			IF F_AxisIsCalibrated(StateDWord := Axis.NcToPlc.StateDWord) THEN
				Done 	:= TRUE;
			ELSE
				Error 	:= TRUE;
				ErrorID := MC_ERROR_CALIBRATION_ERROR; (* functional/calibration error *)
			END_IF;
			iSubState := 0;
		END_IF;
		IF F_AxisInErrorState(StateDWord := Axis.NcToPlc.StateDWord) THEN
			Done := FALSE;
			Error := TRUE;
			ErrorID := Axis.NcToPlc.ErrorCode; (* runtime errorcode *)
			iSubState := 0;
		END_IF;

	9 :	(* read homing position - 2009-04-17 KSt added *)
		fbAdsReadRefPos(	NETID:= TcMcGlobal.NCNETID_TCMC,
							PORT:= TcMcGlobal.NCPORT_TCMC,
							IDXGRP:=TcMcGlobal.Axis.Parameter.IDXGRP+Axis.NcToPlc.AxisId,
							IDXOFFS:= TcMcGlobal.Axis.Parameter.IDXOFFS.REF_POS,
							LEN:= SIZEOF(NcHomePosition),
							DESTADDR:= ADR(NcHomePosition),
							READ:= TRUE,
							TMOUT:= TcMcGlobal.tADSTimeOut);
		IF NOT fbAdsReadRefPos.Busy THEN
			IF fbAdsReadRefPos.Err	THEN
				Error := fbAdsReadRefPos.ERR;
				ErrorID := fbAdsReadRefPos.ERRID;
				iSubState := 0;
			ELSE
				fbSetPosition.Position := NcHomePosition;
				iSubState := iSubState + 1; (* set actual position *)
			END_IF
		END_IF

	10 :	(* Static Homing forcing position from user reference *)
		fbSetPosition.Options.ClearPositionLag:= Options.ClearPositionLag;	(* 2009-04-17 KSt - changed from TRUE to option flag*)
		fbSetPosition(
			Execute:= TRUE,
			(* Position:= Position, 2009-04-17 KSt - must be set before *)
			Mode:= FALSE,	(* absolute mode *)
			Axis:= Axis );
		IF fbSetPosition.Done THEN
			iSubState := iSubState + 1;	(* set reference flag *)
		ELSIF NOT fbSetPosition.Busy THEN
			Error := TRUE;
			ErrorID := fbSetPosition.ErrorID;
			iSubState := 0;
		END_IF

	11 : 	(* Absolute homing - Set reference flag *)
		fbAdsWriteCmd(	NETID:= TcMcGlobal.NCNETID_TCMC,
						PORT:= AMSPORT_R0_NCSAF,
						IDXGRP:= TcMcGlobal.Axis.Functions.IDXGRP+Axis.NcToPlc.AxisId,
						IDXOFFS:= TcMcGlobal.Axis.Functions.IDXOFFS.SETCALFLAG,
						LEN:= SIZEOF(ReferenceFlagValue),
						SRCADDR:= ADR(ReferenceFlagValue),
						WRITE:= TRUE,
						TMOUT:= TcMcGlobal.tADSTimeOut );
		IF NOT fbAdsWriteCmd.Busy THEN
			Error := fbAdsWriteCmd.ERR;
			ErrorID := fbAdsWriteCmd.ERRID;
			Done := NOT Error;
			iSubState := 0;
		END_IF

	ELSE (* CASE : Unknown program state *)
		Error := TRUE;
		ErrorID := 16#FFFFFFFF;
		iSubState := 0;
END_CASE

ADSbusy := fbAdsWriteCmd.BUSY OR fbAdsWriteRefPos.BUSY;

IF iSubState=0 THEN
	(* reset Busy immediately  when sequence ends *)
	IF Busy THEN
		LastExecutionResult.Done := Done;
		LastExecutionResult.CommandAborted := CommandAborted;
		LastExecutionResult.Error := Error;
		LastExecutionResult.ErrorID := ErrorID;
	END_IF
	Busy := FALSE;
ELSE
	(* copy calibration cam to interface *)
	Axis.PlcToNc.ControlDWord.5 := bCalibrationCam;
END_IF

Active := Busy;
END_FUNCTION_BLOCK

(* POU MC_SetPosition, ST *)
FUNCTION_BLOCK MC_SetPosition
(*
	This Function Block shifts the coordinate system of an axis by manipulating both 
	the set-point position as well as the actual position of an axis with the same value 
	without any movement caused. (Re-calibration with same following error).
	This can be used for instance for a reference situation. This Function Block can 
	also be used during motion without changing the commanded position, which is 
	now positioned in the shifted coordinate system.

	Note:
	‘Relative’ means that ‘Position’ is added to the actual position value of the axis 
	at the time of execution. This results in a recalibration by a specified distance. 
	‘Absolute’ means that the actual position value of the axis is set to the value
	specified in the ‘Position’ parameter.
*)
VAR_IN_OUT
	Axis			:	AXIS_REF;	(* B *)	(* Identifies the axis to work upon *)
END_VAR
VAR_INPUT
	Execute		:	BOOL;		(* B *)	(* Start setting position in axis *)
	Position		:	LREAL;		(* B *)	(* Position unit [u] (Means ‘Distance’ if Mode = RELATIVE) *)
	Mode (*Relative*)	: BOOL;		(* E *)	(* RELATIVE =True, ABSOLUTE = False (Default) *)
(* 	MC_ExecutionMode : ENUM *)	(* E *)	(* not available *)
	Options		:	ST_SetPositionOptions;	(* V *)	(* Beckhoff proprietary input *)
END_VAR
VAR_OUTPUT
	Done		:	BOOL;		(* B *)	(* Position has new value *)
	Busy		:	BOOL;		(* E *)	(* Shows that the Function Block is not finished *)
	Error		:	BOOL;		(* B *)	(* Signals that an error has occurred within the Function Block *)
	ErrorID		:	UDINT;		(* E *)	(* Error identification *)
END_VAR
(*
	Note:
	RELATIVE means that Position is added to the actual position value of the axis 
	at the time of execution. This results in a recalibration by a specified distance. 
	ABSOLUTE means that the actual position value of the axis is set to the value 
	specified in the Position parameter.
	When changing the position on the fly, RELATIVE mode is supposed to be preferred
*)
VAR
	ADSbusy	: 	BOOL;
	stSetPos		:	_ST_TcNC_SetPosOnTheFly;
	iState		:	_E_TcMC_STATES := STATE_INITIALIZATION;
	fbAdsWrite	:	ADSWRITE;
END_VAR
{library private}
VAR
	fbOnTrigger	:	R_TRIG;
END_VAR
(*
	PlcOpen comment to MC_SetPosition
		The >Mode< input has later been renamed to >Relative<. Beckhoff cannot change the name for compatibility reasons.
		The input >MC_ExecutionMode<, defined by PlcOpen, is not implemented.
*)

fbOnTrigger(CLK:= Execute);

CASE iState OF
STATE_INITIALIZATION:
	Busy := FALSE;
	IF NOT Execute THEN
		Done := FALSE;
		Error := FALSE;			(* reset at falling edge of Execute *)
		ErrorID := 0;
	END_IF
	IF fbOnTrigger.Q THEN
		Busy := TRUE;
		(* initialize output values *)
		Done := FALSE;
		Error := FALSE;
		ErrorID := 0;
		fbAdsWrite(WRITE := FALSE);

		(* fill structure*)
		stSetPos.fNewActualPos := Position;
		stSetPos.nCtrlDWord.0 := SEL( Options.ClearPositionLag, FALSE, TRUE ); 		(* set bit 0 to clear the lag *)
		stSetPos.nCtrlDWord.1 := SEL( Options.SelectEncoderIndex, FALSE, TRUE ); 	(* set bit 1 to explicitly select an encoder / control loop - KSt 2009-04-09 *)
		stSetPos.nReserved[1]:=0;
		stSetPos.nReserved[2]:=0;

		IF Mode THEN
			(* relative mode *)
			stSetPos.nPosSetType := TCNC_POSSETTYPE_RELATIVE;
			stSetPos.fPreviousActualPos := 0;	(* value not used any longer since 2009-01-28 *)
		ELSE
			(* absolute mode *)
			stSetPos.nPosSetType := TCNC_POSSETTYPE_ABSOLUTE;
			stSetPos.fPreviousActualPos := Axis.NcToPlc.ActPos;	(* value not used any longer since 2009-01-28 *)
		END_IF

		IF Options.SelectEncoderIndex THEN (* KSt 2009-04-09 *)
			(* select the user defined encoder/control loop explicitly *)
			fbAdsWrite.IDXOFFS:= TcMcGlobal.Axis.Functions.IDXOFFS.SETPOSONTHEFLY + Options.EncoderIndex * 16#00100000;
		ELSE
			(* select the encoder / control loop that is defined by the AXIS_REF interface
				0  	=  select active encoder / control loop		- used when standard AXIS_REF interface is used
				1..n 	=  explicit encoder / control loop selection 	- used when dedicated encoder AXIS_REF interface is used 		*)
			fbAdsWrite.IDXOFFS:= TcMcGlobal.Axis.Functions.IDXOFFS.SETPOSONTHEFLY + Axis.NcToPlc.ControlLoopIndex * 16#00100000;
		END_IF

		fbAdsWrite(	NETID:= TcMcGlobal.NCNETID_TCMC,
					PORT:= AMSPORT_R0_NCSAF,
					IDXGRP:=TcMcGlobal.Axis.Functions.IDXGRP + Axis.NcToPlc.AxisId,
(*					IDXOFFS:= TcMcGlobal.Axis.Functions.IDXOFFS.SETPOSONTHEFLY + Options.EncoderIndex * 16#100000, *)(* add sub index - KSt 2008-10-22 *)
(*					IDXOFFS:= TcMcGlobal.Axis.Functions.IDXOFFS.SETPOSONTHEFLY, *)	(* see selection above - KSt 2009-04-09 *)
					LEN:= SIZEOF(stSetPos),
					SRCADDR:= ADR(stSetPos),
					WRITE:= TRUE,
					TMOUT:= TcMcGlobal.tADSTimeOut);
		iState := STATE_ORDER;
	END_IF;

STATE_ORDER:
	fbAdsWrite();
	IF NOT fbAdsWrite.Busy THEN
		IF fbAdsWrite.Err THEN
			ErrorID := fbAdsWrite.ErrId;
			Error := TRUE;
		ELSE
			Done := TRUE;
		END_IF;
		fbAdsWrite(WRITE := FALSE);
		iState := STATE_INITIALIZATION;
	END_IF;

ELSE  (* CASE : Unknown program state *)
	Error := TRUE;
	ErrorID := 16#FFFFFFFF;
	iState:= STATE_INITIALIZATION;
END_CASE

ADSbusy := fbAdsWrite.BUSY;

IF iState=STATE_INITIALIZATION THEN
	(* reset Busy immediately  when sequence ends *)
	Busy := FALSE;
END_IF
END_FUNCTION_BLOCK

(* POU MC_Jog, ST *)
FUNCTION_BLOCK MC_Jog
(*	This function block commands a jogged movement to an axis.*)
VAR_IN_OUT
	Axis				:	AXIS_REF;
END_VAR
VAR_INPUT
	JogForward 		: 	BOOL;
	JogBackwards 	: 	BOOL;
	Mode			: 	E_JogMode;
	Position 			: 	LREAL;
	Velocity			:	LREAL;
	Acceleration		:	LREAL;
	Deceleration		:	LREAL;
	Jerk				:	LREAL;
(*	BufferMode		:	MC_BufferMode;*)(* E *)
END_VAR
VAR_OUTPUT
	Done			:	BOOL;
	Busy 			:	BOOL;
	Active 			:	BOOL;
	CommandAborted	:	BOOL;
	Error			:	BOOL;
	ErrorID			:	UDINT;
END_VAR
VAR
	state: INT;
	LastExecutionResult: _ST_FunctionBlockResults;
	StateDWord: BOOL;
END_VAR
{library private}
VAR
	ExecuteMoveVelocity: BOOL;
	MoveVelocity: MC_MoveVelocity;
	MoveVelocityOut : ST_McOutputs;
	Direction: MC_Direction;

	ExecuteHalt: BOOL;
	Halt: MC_Halt;
	HaltOut : ST_McOutputs;

	ExecuteMoveAbsolute: BOOL;
	MoveAbsolute: MC_MoveAbsolute;
	MoveAbsoluteOut : ST_McOutputs;

	ExecuteMoveRelative: BOOL;
	MoveRelative : MC_MoveRelative;
	MoveRelativeOut : ST_McOutputs;

	JogMove: _FB_MoveUniversalGeneric;
	LastJogMoveResult: _ST_FunctionBlockResults;
	ExecuteJogMove: BOOL;
	StartType: _E_TCNC_StartPosType;
	JogMoveOut : ST_McOutputs;

	JogEnd: BOOL;
	TargetPosition: LREAL;
	modulo: LREAL;
END_VAR
ActCheckJogEnd();

CASE state OF
	0 : (* Initialization *)
		Busy := FALSE;
		Active := FALSE;
		ExecuteMoveVelocity := FALSE;
		ExecuteMoveRelative := FALSE;
		ExecuteMoveAbsolute := FALSE;
		ExecuteJogMove := FALSE;
		ExecuteHalt := FALSE;

		IF NOT JogForward AND NOT JogBackwards THEN (* 2009-03-12 *)
			Done := FALSE;
			CommandAborted := FALSE;
			Error := FALSE;
			ErrorID := 0;
		ELSIF (JogForward OR JogBackwards) AND F_AxisInProtectedMode(Axis.NcToPlc.StateDWord) THEN(* 2009-11-18 KSt *)
			(* MC_Jog cannot be used in protected mode (e. g. slave axis) *)
			Error := TRUE;
			ErrorID := MC_ERROR_AXIS_IN_PROTECTED_MODE;
		ELSIF JogForward AND NOT JogBackwards THEN
			Done := FALSE;
			Busy := TRUE;
			CommandAborted := FALSE;
			Error := FALSE;
			ErrorID := 0;
			Direction := MC_Positive_Direction;
			CASE Mode OF
				MC_JOGMODE_STANDARD_SLOW :
					StartType := TCNC_START_ENDLESSPLUS_SLOWMANUAL;
					ExecuteJogMove := TRUE;
					state := 3;
				MC_JOGMODE_STANDARD_FAST :
					StartType := TCNC_START_ENDLESSPLUS_FASTMANUAL;
					ExecuteJogMove := TRUE;
					state := 3;
				MC_JOGMODE_CONTINOUS :
					ExecuteMoveVelocity := TRUE;
					state := 1;
				MC_JOGMODE_INCHING :
					TargetPosition := Position;
					ExecuteMoveRelative := TRUE;
					state := 4;
				MC_JOGMODE_INCHING_MODULO :
					TargetPosition := Axis.NcToPlc.SetPos - Axis.NcToPlc.ModuloSetPos + Position;
					ExecuteMoveAbsolute := TRUE;
					state := 2;
			ELSE
				Busy := FALSE;
			END_CASE
		ELSIF JogBackwards AND NOT JogForward THEN
			Done := FALSE;
			Busy := TRUE;
			CommandAborted := FALSE;
			Error := FALSE;
			ErrorID := 0;
			Direction := MC_Negative_Direction;
			CASE Mode OF
				MC_JOGMODE_STANDARD_SLOW :
					StartType := TCNC_START_ENDLESSMINUS_SLOWMANUAL;
					ExecuteJogMove := TRUE;
					state := 3;
				MC_JOGMODE_STANDARD_FAST :
					StartType := TCNC_START_ENDLESSMINUS_FASTMANUAL;
					ExecuteJogMove := TRUE;
					state := 3;
				MC_JOGMODE_CONTINOUS :
					ExecuteMoveVelocity := TRUE;
					state := 1;
				MC_JOGMODE_INCHING :
					TargetPosition := - Position;
					ExecuteMoveRelative := TRUE;
					state := 4;
				MC_JOGMODE_INCHING_MODULO :
					modulo := Axis.NcToPlc.ModuloSetPos;
					IF modulo = 0 THEN
						TargetPosition := Axis.NcToPlc.SetPos - Position;
					ELSE
						TargetPosition := Axis.NcToPlc.SetPos - Axis.NcToPlc.ModuloSetPos;
					END_IF
					ExecuteMoveAbsolute := TRUE;
					state := 2;
			ELSE
				Busy := FALSE;
			END_CASE
		END_IF

	1 : (* continous jogging with MoveVelocity *)
		IF JogEnd THEN
			ExecuteMoveVelocity := FALSE;
			ExecuteHalt := TRUE;
		END_IF
		IF NOT MoveVelocity.Busy AND NOT Halt.Busy AND NOT F_AxisHasJob(Axis.NcToPlc.StateDWord) THEN
			Error := MoveVelocity.Error OR Halt.Error OR F_AxisInErrorState(Axis.NcToPlc.StateDWord);
			ErrorID := SEL( F_AxisInErrorState(Axis.NcToPlc.StateDWord), SEL(MoveVelocity.Error, Halt.ErrorID, MoveVelocity.ErrorID ), Axis.NcToPlc.ErrorCode);
			CommandAborted := NOT Error AND MoveVelocity.CommandAborted AND NOT ExecuteHalt; (* logic fixed 14.3.07 KSt *)
			Done := NOT Error AND NOT CommandAborted;
			ExecuteMoveVelocity := FALSE;
			ExecuteHalt := FALSE;
			IF JogEnd OR Done THEN
				state := 0;
			ELSE
				state := 9;
			END_IF
		END_IF

	2 : (* inching with MoveAbsolute *)
		IF 	Done OR
			(NOT MoveAbsolute.Busy AND NOT F_AxisHasJob(Axis.NcToPlc.StateDWord)) THEN
			Error := MoveAbsolute.Error;
			ErrorID := MoveAbsolute.ErrorID;
			CommandAborted := MoveAbsolute.CommandAborted;
			Done := NOT Error AND NOT CommandAborted;
			ExecuteMoveAbsolute := FALSE;
			IF JogEnd THEN
				state := 0;
			ELSE
				state := 9;
			END_IF
		END_IF

	3 : (* continous jogging with system parameters *)
		IF JogEnd THEN
			ExecuteJogMove := FALSE;
			ExecuteHalt := TRUE;
		END_IF
		IF NOT JogMove.Busy AND NOT Halt.Busy AND NOT F_AxisHasJob(Axis.NcToPlc.StateDWord) THEN
			Error := JogMove.Error OR Halt.Error OR F_AxisInErrorState(Axis.NcToPlc.StateDWord);
			ErrorID := SEL( F_AxisInErrorState(Axis.NcToPlc.StateDWord), SEL(JogMove.Error, Halt.ErrorID, JogMove.ErrorID ), Axis.NcToPlc.ErrorCode);
			CommandAborted := NOT Error AND JogMove.CommandAborted AND NOT ExecuteHalt; (* logic fixed 14.3.07 KSt *)
			Done := NOT Error AND NOT CommandAborted;
			ExecuteJogMove := FALSE;
			ExecuteHalt := FALSE;
			IF JogEnd OR Done THEN
				state := 0;
			ELSE
				state := 9;
			END_IF
		END_IF

	4 : (* inching with MoveRelative *)
		IF 	Done OR
			(NOT MoveRelative.Busy AND NOT F_AxisHasJob(Axis.NcToPlc.StateDWord)) THEN
			Error := MoveRelative.Error;
			ErrorID := MoveRelative.ErrorID;
			CommandAborted := MoveRelative.CommandAborted;
			Done := NOT Error AND NOT CommandAborted;
			ExecuteMoveRelative := FALSE;
			IF JogEnd THEN
				state := 0;
			ELSE
				state := 9;
			END_IF
		END_IF

	9 :	(* wait for falling edge on execute *)
		IF JogEnd THEN
			state := 0;
		END_IF
END_CASE

ActJogMove();

